Universal Robots URScript: test_regenerated.script

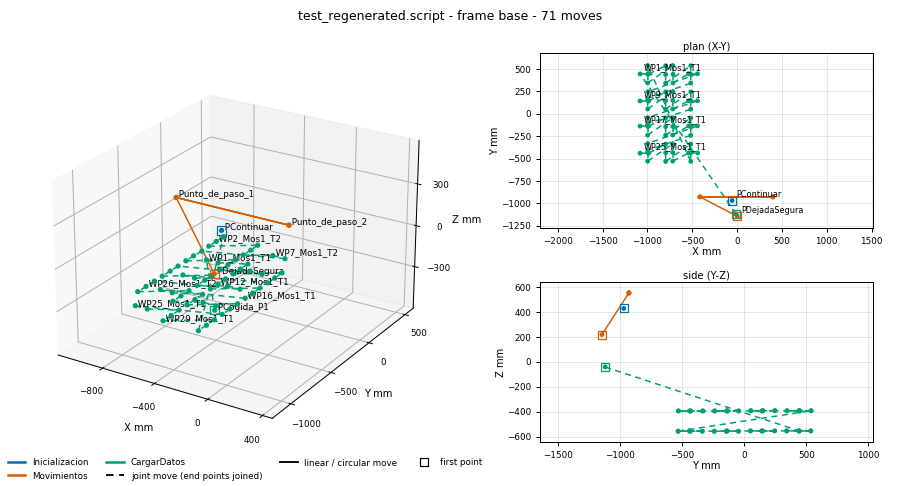
[picture p0: tool path of test_regenerated.script in frame base, 71 of 89 moves have a stored position in this frame; points joined in program order, loops and branches not executed]
def P002_008_L16_REC_AMB_MF():
  set_safety_mode_transition_hardness(1)
  set_tool_communication(False, 115200, 0, 1, 1.5, 3.5)
  set_tool_output_mode(0)
  set_tool_digital_output_mode(0, 1)
  set_tool_digital_output_mode(1, 1)
  set_tool_voltage(24)
  set_tcp(p[0.0,-0.14,0.054,0.0,0.0,0.0])
  set_payload(0.84)
  set_standard_analog_input_domain(0, 1)
  set_standard_analog_input_domain(1, 1)
  set_tool_analog_input_domain(0, 1)
  set_tool_analog_input_domain(1, 1)
  set_analog_outputdomain(0, 0)
  set_analog_outputdomain(1, 0)
  set_input_actions_to_default()
  set_runstate_gp_boolean_output_to_value(15, 3)
  set_gravity([0.0, 0.0, 9.82])
  step_count_91e529f0_9954_4772_b49d_1590ab779229 = 0
  thread Step_Counter_Thread_984ad8c2_81a8_4544_ae12_e3986bad7eaf():
    while (True):
      step_count_91e529f0_9954_4772_b49d_1590ab779229 = step_count_91e529f0_9954_4772_b49d_1590ab779229 + 1
      sync()
    end
  end
  run Step_Counter_Thread_984ad8c2_81a8_4544_ae12_e3986bad7eaf()
  global AlarmaVF2=False
  global ordenM9_T1=[1, 2, 3, 4, 5, 6, 7, 8, 1, 1, 1, 1, 1, 1, 1, 1, 1, 1, 1, 1, 1, 1, 1, 1, 1]
  global AlarmaVF1=False
  global linea=1
  global AlarmaQM2=False
  global LineaHabilitada=[True, True]
  global AlarmaQM1=False
  global ContPrd=0
  global P_Tipo1_Mos9=[p[100, 100, 100, 0, 0, 0], p[100, 100, 100, 0, 0, 0], p[100, 100, 100, 0, 0, 0], p[100, 100, 100, 0, 0, 0], p[100, 100, 100, 0, 0, 0], p[100, 100, 100, 0, 0, 0], p[100, 100, 100, 0, 0, 0], p[100, 100, 100, 0, 0, 0], p[100, 100, 100, 0, 0, 0], p[100, 100, 100, 0, 0, 0], p[100, 100, 100, 0, 0, 0], p[100, 100, 100, 0, 0, 0], p[100, 100, 100, 0, 0, 0], p[100, 100, 100, 0, 0, 0], p[100, 100, 100, 0, 0, 0], p[100, 100, 100, 0, 0, 0], p[100, 100, 100, 0, 0, 0], p[100, 100, 100, 0, 0, 0], p[100, 100, 100, 0, 0, 0], p[100, 100, 100, 0, 0, 0], p[100, 100, 100, 0, 0, 0], p[100, 100, 100, 0, 0, 0], p[100, 100, 100, 0, 0, 0], p[100, 100, 100, 0, 0, 0], p[100, 100, 100, 0, 0, 0]]
  global P_Tipo1_Mos8=[p[100, 100, 100, 0, 0, 0], p[100, 100, 100, 0, 0, 0], p[100, 100, 100, 0, 0, 0], p[100, 100, 100, 0, 0, 0], p[100, 100, 100, 0, 0, 0], p[100, 100, 100, 0, 0, 0], p[100, 100, 100, 0, 0, 0], p[100, 100, 100, 0, 0, 0], p[100, 100, 100, 0, 0, 0], p[100, 100, 100, 0, 0, 0], p[100, 100, 100, 0, 0, 0], p[100, 100, 100, 0, 0, 0], p[100, 100, 100, 0, 0, 0], p[100, 100, 100, 0, 0, 0], p[100, 100, 100, 0, 0, 0], p[100, 100, 100, 0, 0, 0], p[100, 100, 100, 0, 0, 0], p[100, 100, 100, 0, 0, 0], p[100, 100, 100, 0, 0, 0], p[100, 100, 100, 0, 0, 0], p[100, 100, 100, 0, 0, 0], p[100, 100, 100, 0, 0, 0], p[100, 100, 100, 0, 0, 0], p[100, 100, 100, 0, 0, 0], p[100, 100, 100, 0, 0, 0]]
  global P_Tipo1_Mos7=[p[100, 100, 100, 0, 0, 0], p[100, 100, 100, 0, 0, 0], p[100, 100, 100, 0, 0, 0], p[100, 100, 100, 0, 0, 0], p[100, 100, 100, 0, 0, 0], p[100, 100, 100, 0, 0, 0], p[100, 100, 100, 0, 0, 0], p[100, 100, 100, 0, 0, 0], p[100, 100, 100, 0, 0, 0], p[100, 100, 100, 0, 0, 0], p[100, 100, 100, 0, 0, 0], p[100, 100, 100, 0, 0, 0], p[100, 100, 100, 0, 0, 0], p[100, 100, 100, 0, 0, 0], p[100, 100, 100, 0, 0, 0], p[100, 100, 100, 0, 0, 0], p[100, 100, 100, 0, 0, 0], p[100, 100, 100, 0, 0, 0], p[100, 100, 100, 0, 0, 0], p[100, 100, 100, 0, 0, 0], p[100, 100, 100, 0, 0, 0], p[100, 100, 100, 0, 0, 0], p[100, 100, 100, 0, 0, 0], p[100, 100, 100, 0, 0, 0], p[100, 100, 100, 0, 0, 0]]
  global P_Tipo1_Mos6=[p[100, 100, 100, 0, 0, 0], p[100, 100, 100, 0, 0, 0], p[100, 100, 100, 0, 0, 0], p[100, 100, 100, 0, 0, 0], p[100, 100, 100, 0, 0, 0], p[100, 100, 100, 0, 0, 0], p[100, 100, 100, 0, 0, 0], p[100, 100, 100, 0, 0, 0], p[100, 100, 100, 0, 0, 0], p[100, 100, 100, 0, 0, 0], p[100, 100, 100, 0, 0, 0], p[100, 100, 100, 0, 0, 0], p[100, 100, 100, 0, 0, 0], p[100, 100, 100, 0, 0, 0], p[100, 100, 100, 0, 0, 0], p[100, 100, 100, 0, 0, 0], p[100, 100, 100, 0, 0, 0], p[100, 100, 100, 0, 0, 0], p[100, 100, 100, 0, 0, 0], p[100, 100, 100, 0, 0, 0], p[100, 100, 100, 0, 0, 0], p[100, 100, 100, 0, 0, 0], p[100, 100, 100, 0, 0, 0], p[100, 100, 100, 0, 0, 0], p[100, 100, 100, 0, 0, 0]]
  global P_Tipo1_Mos5=[p[100, 100, 100, 0, 0, 0], p[100, 100, 100, 0, 0, 0], p[100, 100, 100, 0, 0, 0], p[100, 100, 100, 0, 0, 0], p[100, 100, 100, 0, 0, 0], p[100, 100, 100, 0, 0, 0], p[100, 100, 100, 0, 0, 0], p[100, 100, 100, 0, 0, 0], p[100, 100, 100, 0, 0, 0], p[100, 100, 100, 0, 0, 0], p[100, 100, 100, 0, 0, 0], p[100, 100, 100, 0, 0, 0], p[100, 100, 100, 0, 0, 0], p[100, 100, 100, 0, 0, 0], p[100, 100, 100, 0, 0, 0], p[100, 100, 100, 0, 0, 0], p[100, 100, 100, 0, 0, 0], p[100, 100, 100, 0, 0, 0], p[100, 100, 100, 0, 0, 0], p[100, 100, 100, 0, 0, 0], p[100, 100, 100, 0, 0, 0], p[100, 100, 100, 0, 0, 0], p[100, 100, 100, 0, 0, 0], p[100, 100, 100, 0, 0, 0], p[100, 100, 100, 0, 0, 0]]
  global P_Tipo1_Mos4=[p[100, 100, 100, 0, 0, 0], p[100, 100, 100, 0, 0, 0], p[100, 100, 100, 0, 0, 0], p[100, 100, 100, 0, 0, 0], p[100, 100, 100, 0, 0, 0], p[100, 100, 100, 0, 0, 0], p[100, 100, 100, 0, 0, 0], p[100, 100, 100, 0, 0, 0], p[100, 100, 100, 0, 0, 0], p[100, 100, 100, 0, 0, 0], p[100, 100, 100, 0, 0, 0], p[100, 100, 100, 0, 0, 0], p[100, 100, 100, 0, 0, 0], p[100, 100, 100, 0, 0, 0], p[100, 100, 100, 0, 0, 0], p[100, 100, 100, 0, 0, 0], p[100, 100, 100, 0, 0, 0], p[100, 100, 100, 0, 0, 0], p[100, 100, 100, 0, 0, 0], p[100, 100, 100, 0, 0, 0], p[100, 100, 100, 0, 0, 0], p[100, 100, 100, 0, 0, 0], p[100, 100, 100, 0, 0, 0], p[100, 100, 100, 0, 0, 0], p[100, 100, 100, 0, 0, 0]]
  global PrdsReq=1
  global P_Tipo1_Mos3=[p[1.16604, 0.55562, 0.63575, 3.14108, -0.00276, -8.40000000000000035E-04], p[0.94603, 0.55481, 0.62022, 3.14109, -0.00285, -8.89999999999999949E-04], p[0.72803, 0.55407, 0.62302, 3.1411, -0.01338, -8.19999999999999982E-04], p[0.511, 0.5552, 0.61604, 3.14122, -0.01324, -8.49999999999999953E-04], p[0.29303, 0.5544, 0.62251, 3.14118, -0.01329, -8.99999999999999975E-04], p[1.00128, 0.17498, 0.62283, 2.22765, -2.21424, -2.30000000000000007E-04], p[0.4544, 0.17301, 0.61254, 2.22767, -2.21422, -2.99999999999999974E-04], p[100, 100, 100, 0, 0, 0], p[100, 100, 100, 0, 0, 0], p[100, 100, 100, 0, 0, 0], p[100, 100, 100, 0, 0, 0], p[100, 100, 100, 0, 0, 0], p[100, 100, 100, 0, 0, 0], p[100, 100, 100, 0, 0, 0], p[100, 100, 100, 0, 0, 0], p[100, 100, 100, 0, 0, 0], p[100, 100, 100, 0, 0, 0], p[100, 100, 100, 0, 0, 0], p[100, 100, 100, 0, 0, 0], p[100, 100, 100, 0, 0, 0], p[100, 100, 100, 0, 0, 0], p[100, 100, 100, 0, 0, 0], p[100, 100, 100, 0, 0, 0], p[100, 100, 100, 0, 0, 0], p[100, 100, 100, 0, 0, 0]]
  global P_Tipo1_Mos2=[p[0.99704, 0.69994, 0.4025, 2.20418, 2.23837, -0.00134], p[0.99871, 0.49941, 0.39482, 2.21365, 2.229, -0.00133], p[0.70631, 0.6015, 0.38963, 0.00568, -3.14107, 0.00118], p[0.50788, 0.60078, 0.39072, 0.00568, -3.14107, 0.00118], p[0.30863, 0.60101, 0.39721, 0.00568, -3.14107, 0.00118], p[0.10677, 0.60171, 0.39277, 0.00568, -3.14107, 0.00118], p[1.0952, 0.20925, 0.39062, 3.14092, 0.00568, -7.10000000000000019E-04], p[0.89523, 0.21023, 0.40246, 3.14092, 0.00568, -7.10000000000000019E-04], p[0.6952, 0.21273, 0.39826, 3.14092, 0.00568, -7.10000000000000019E-04], p[0.49709, 0.21201, 0.39756, 3.14092, 0.00568, -7.10000000000000019E-04], p[0.20516, 0.31346, 0.39069, 2.22486, -2.21683, 2.99999999999999974E-04], p[0.20589, 0.11488, 0.39661, 2.22486, -2.21683, 2.99999999999999974E-04], p[100, 100, 100, 0, 0, 0], p[100, 100, 100, 0, 0, 0], p[100, 100, 100, 0, 0, 0], p[100, 100, 100, 0, 0, 0], p[100, 100, 100, 0, 0, 0], p[100, 100, 100, 0, 0, 0], p[100, 100, 100, 0, 0, 0], p[100, 100, 100, 0, 0, 0], p[100, 100, 100, 0, 0, 0], p[100, 100, 100, 0, 0, 0], p[100, 100, 100, 0, 0, 0], p[100, 100, 100, 0, 0, 0], p[100, 100, 100, 0, 0, 0]]
  global PalletOk=[True, False]
  global P_Tipo1_Mos1=[p[1.04122, 0.73691, 0.32186, -3.1356, -0.00672, -0.01102], p[1.04157, 0.63991, 0.32193, -3.1356, -0.00674, -0.01104], p[1.13376, 0.45174, 0.32215, -2.21965, 2.21023, -0.00123], p[1.03676, 0.45138, 0.32217, -2.21965, 2.21026, -0.00124], p[0.93976, 0.451, 0.3222, -2.21964, 2.21028, -0.00128], p[1.13477, 0.17175, 0.32228, -2.21961, 2.21034, -0.00133], p[1.03777, 0.1714, 0.32233, -2.21962, 2.21032, -0.00135], p[0.94077, 0.17108, 0.32239, -2.21962, 2.21028, -0.00136], p[0.73923, 0.73581, 0.32199, -3.13562, -0.00685, -0.01105], p[0.73959, 0.63882, 0.32205, -3.13564, -0.00684, -0.01107], p[0.84276, 0.45068, 0.32225, -2.21963, 2.21023, -0.00125], p[0.74576, 0.45033, 0.32229, -2.21964, 2.21024, -0.00125], p[0.64876, 0.44998, 0.32233, -2.21967, 2.21024, -0.00121], p[0.84377, 0.17069, 0.32246, -2.2197, 2.21021, -0.00117], p[0.74677, 0.17036, 0.32253, -2.21965, 2.2102, -0.00112], p[0.64977, 0.17002, 0.32257, -2.21967, 2.21018, -0.00108], p[0.45923, 0.73477, 0.32211, -3.13566, -0.00681, -0.01102], p[0.45959, 0.63781, 0.32216, -3.13571, -0.00678, -0.01101], p[0.55176, 0.44964, 0.32025, 2.216, 2.22572, 0.01433], p[0.45476, 0.4493, 0.3203, 2.21603, 2.22569, 0.01434], p[0.35776, 0.44894, 0.32035, 2.21598, 2.22574, 0.01432], p[0.55277, 0.16964, 0.32047, 2.21602, 2.22572, 0.0143], p[0.45577, 0.16927, 0.3205, 2.21599, 2.22573, 0.0143], p[0.35877, 0.16893, 0.32054, 2.21602, 2.2257, 0.0143], p[0.15723, 0.73362, 0.3222, -3.13576, -0.00684, -0.01106]]
  global NPaletTot=5422
  global PalletReady=[True, True]
  global Rec_AltoPrd=[160, 160, 0, 0, 0, 0, 0, 0, 0, 0]
  global P_Tipo2_Mos9=[p[100, 100, 100, 0, 0, 0], p[100, 100, 100, 0, 0, 0], p[100, 100, 100, 0, 0, 0], p[100, 100, 100, 0, 0, 0], p[100, 100, 100, 0, 0, 0], p[100, 100, 100, 0, 0, 0], p[100, 100, 100, 0, 0, 0], p[100, 100, 100, 0, 0, 0], p[100, 100, 100, 0, 0, 0], p[100, 100, 100, 0, 0, 0], p[100, 100, 100, 0, 0, 0], p[100, 100, 100, 0, 0, 0], p[100, 100, 100, 0, 0, 0], p[100, 100, 100, 0, 0, 0], p[100, 100, 100, 0, 0, 0], p[100, 100, 100, 0, 0, 0], p[100, 100, 100, 0, 0, 0], p[100, 100, 100, 0, 0, 0], p[100, 100, 100, 0, 0, 0], p[100, 100, 100, 0, 0, 0], p[100, 100, 100, 0, 0, 0], p[100, 100, 100, 0, 0, 0], p[100, 100, 100, 0, 0, 0], p[100, 100, 100, 0, 0, 0], p[100, 100, 100, 0, 0, 0]]
  global P_Tipo2_Mos8=[p[100, 100, 100, 0, 0, 0], p[100, 100, 100, 0, 0, 0], p[100, 100, 100, 0, 0, 0], p[100, 100, 100, 0, 0, 0], p[100, 100, 100, 0, 0, 0], p[100, 100, 100, 0, 0, 0], p[100, 100, 100, 0, 0, 0], p[100, 100, 100, 0, 0, 0], p[100, 100, 100, 0, 0, 0], p[100, 100, 100, 0, 0, 0], p[100, 100, 100, 0, 0, 0], p[100, 100, 100, 0, 0, 0], p[100, 100, 100, 0, 0, 0], p[100, 100, 100, 0, 0, 0], p[100, 100, 100, 0, 0, 0], p[100, 100, 100, 0, 0, 0], p[100, 100, 100, 0, 0, 0], p[100, 100, 100, 0, 0, 0], p[100, 100, 100, 0, 0, 0], p[100, 100, 100, 0, 0, 0], p[100, 100, 100, 0, 0, 0], p[100, 100, 100, 0, 0, 0], p[100, 100, 100, 0, 0, 0], p[100, 100, 100, 0, 0, 0], p[100, 100, 100, 0, 0, 0]]
  global P_Tipo2_Mos7=[p[100, 100, 100, 0, 0, 0], p[100, 100, 100, 0, 0, 0], p[100, 100, 100, 0, 0, 0], p[100, 100, 100, 0, 0, 0], p[100, 100, 100, 0, 0, 0], p[100, 100, 100, 0, 0, 0], p[100, 100, 100, 0, 0, 0], p[100, 100, 100, 0, 0, 0], p[100, 100, 100, 0, 0, 0], p[100, 100, 100, 0, 0, 0], p[100, 100, 100, 0, 0, 0], p[100, 100, 100, 0, 0, 0], p[100, 100, 100, 0, 0, 0], p[100, 100, 100, 0, 0, 0], p[100, 100, 100, 0, 0, 0], p[100, 100, 100, 0, 0, 0], p[100, 100, 100, 0, 0, 0], p[100, 100, 100, 0, 0, 0], p[100, 100, 100, 0, 0, 0], p[100, 100, 100, 0, 0, 0], p[100, 100, 100, 0, 0, 0], p[100, 100, 100, 0, 0, 0], p[100, 100, 100, 0, 0, 0], p[100, 100, 100, 0, 0, 0], p[100, 100, 100, 0, 0, 0]]
  global P_Tipo2_Mos6=[p[100, 100, 100, 0, 0, 0], p[100, 100, 100, 0, 0, 0], p[100, 100, 100, 0, 0, 0], p[100, 100, 100, 0, 0, 0], p[100, 100, 100, 0, 0, 0], p[100, 100, 100, 0, 0, 0], p[100, 100, 100, 0, 0, 0], p[100, 100, 100, 0, 0, 0], p[100, 100, 100, 0, 0, 0], p[100, 100, 100, 0, 0, 0], p[100, 100, 100, 0, 0, 0], p[100, 100, 100, 0, 0, 0], p[100, 100, 100, 0, 0, 0], p[100, 100, 100, 0, 0, 0], p[100, 100, 100, 0, 0, 0], p[100, 100, 100, 0, 0, 0], p[100, 100, 100, 0, 0, 0], p[100, 100, 100, 0, 0, 0], p[100, 100, 100, 0, 0, 0], p[100, 100, 100, 0, 0, 0], p[100, 100, 100, 0, 0, 0], p[100, 100, 100, 0, 0, 0], p[100, 100, 100, 0, 0, 0], p[100, 100, 100, 0, 0, 0], p[100, 100, 100, 0, 0, 0]]
  global P_Tipo2_Mos5=[p[100, 100, 100, 0, 0, 0], p[100, 100, 100, 0, 0, 0], p[100, 100, 100, 0, 0, 0], p[100, 100, 100, 0, 0, 0], p[100, 100, 100, 0, 0, 0], p[100, 100, 100, 0, 0, 0], p[100, 100, 100, 0, 0, 0], p[100, 100, 100, 0, 0, 0], p[100, 100, 100, 0, 0, 0], p[100, 100, 100, 0, 0, 0], p[100, 100, 100, 0, 0, 0], p[100, 100, 100, 0, 0, 0], p[100, 100, 100, 0, 0, 0], p[100, 100, 100, 0, 0, 0], p[100, 100, 100, 0, 0, 0], p[100, 100, 100, 0, 0, 0], p[100, 100, 100, 0, 0, 0], p[100, 100, 100, 0, 0, 0], p[100, 100, 100, 0, 0, 0], p[100, 100, 100, 0, 0, 0], p[100, 100, 100, 0, 0, 0], p[100, 100, 100, 0, 0, 0], p[100, 100, 100, 0, 0, 0], p[100, 100, 100, 0, 0, 0], p[100, 100, 100, 0, 0, 0]]
  global NCapaAct=[1, 1]
  global P_Tipo2_Mos4=[p[100, 100, 100, 0, 0, 0], p[100, 100, 100, 0, 0, 0], p[100, 100, 100, 0, 0, 0], p[100, 100, 100, 0, 0, 0], p[100, 100, 100, 0, 0, 0], p[100, 100, 100, 0, 0, 0], p[100, 100, 100, 0, 0, 0], p[100, 100, 100, 0, 0, 0], p[100, 100, 100, 0, 0, 0], p[100, 100, 100, 0, 0, 0], p[100, 100, 100, 0, 0, 0], p[100, 100, 100, 0, 0, 0], p[100, 100, 100, 0, 0, 0], p[100, 100, 100, 0, 0, 0], p[100, 100, 100, 0, 0, 0], p[100, 100, 100, 0, 0, 0], p[100, 100, 100, 0, 0, 0], p[100, 100, 100, 0, 0, 0], p[100, 100, 100, 0, 0, 0], p[100, 100, 100, 0, 0, 0], p[100, 100, 100, 0, 0, 0], p[100, 100, 100, 0, 0, 0], p[100, 100, 100, 0, 0, 0], p[100, 100, 100, 0, 0, 0], p[100, 100, 100, 0, 0, 0]]
  global P_Tipo2_Mos3=[p[1.00663, 0.71329, 0.77118, 2.22767, -2.21422, -2.99999999999999974E-04], p[0.45784, 0.71261, 0.76931, 2.22767, -2.21422, -2.99999999999999974E-04], p[1.16656, 0.33923, 0.80534, 3.1413, -0.00972, -9.60000000000000024E-04], p[0.9489, 0.33841, 0.79064, 3.14125, -0.01511, -0.00113], p[0.73088, 0.33763, 0.77696, 3.14125, -0.01511, -0.00115], p[0.5119, 0.33683, 0.78134, 3.14126, -0.01514, -0.00122], p[0.29291, 0.33753, 0.79002, 3.14126, -0.0151, -0.00118], p[100, 100, 100, 0, 0, 0], p[100, 100, 100, 0, 0, 0], p[100, 100, 100, 0, 0, 0], p[100, 100, 100, 0, 0, 0], p[100, 100, 100, 0, 0, 0], p[100, 100, 100, 0, 0, 0], p[100, 100, 100, 0, 0, 0], p[100, 100, 100, 0, 0, 0], p[100, 100, 100, 0, 0, 0], p[100, 100, 100, 0, 0, 0], p[100, 100, 100, 0, 0, 0], p[100, 100, 100, 0, 0, 0], p[100, 100, 100, 0, 0, 0], p[100, 100, 100, 0, 0, 0], p[100, 100, 100, 0, 0, 0], p[100, 100, 100, 0, 0, 0], p[100, 100, 100, 0, 0, 0], p[100, 100, 100, 0, 0, 0]]
  global P_Tipo2_Mos2=[p[1.09673, 0.60531, 0.52579, 0.00568, -3.14105, 0.00108], p[0.89826, 0.60459, 0.53036, 0.00568, -3.14105, 0.00108], p[0.69753, 0.60155, 0.53003, 0.00568, -3.14105, 0.00108], p[0.49739, 0.60082, 0.52062, 0.00568, -3.14105, 0.00108], p[0.20624, 0.7039, 0.53456, 2.22483, -2.21679, 2.70000000000000003E-04], p[0.2033, 0.50369, 0.53493, 2.22483, -2.21679, 2.70000000000000003E-04], p[1.00083, 0.30839, 0.52599, 2.21734, 2.22537, -0.00119], p[1.00155, 0.11082, 0.53432, 2.21734, 2.22537, -0.00119], p[0.70593, 0.21094, 0.5328, 3.14079, 0.00568, -6.59999999999999996E-04], p[0.50462, 0.2113, 0.536, 3.14079, 0.00568, -6.59999999999999996E-04], p[0.30453, 0.20978, 0.53196, 3.14079, 0.00568, -6.59999999999999996E-04], p[0.10494, 0.20881, 0.53476, 3.14079, 0.00568, -6.59999999999999996E-04], p[100, 100, 100, 0, 0, 0], p[100, 100, 100, 0, 0, 0], p[100, 100, 100, 0, 0, 0], p[100, 100, 100, 0, 0, 0], p[100, 100, 100, 0, 0, 0], p[100, 100, 100, 0, 0, 0], p[100, 100, 100, 0, 0, 0], p[100, 100, 100, 0, 0, 0], p[100, 100, 100, 0, 0, 0], p[100, 100, 100, 0, 0, 0], p[100, 100, 100, 0, 0, 0], p[100, 100, 100, 0, 0, 0], p[100, 100, 100, 0, 0, 0]]
  global Rec_LargoPrd=[280, 280, 0, 0, 0, 0, 0, 0, 0, 0]
  global P_Tipo2_Mos1=[p[1.13563, 0.65237, 0.48446, -2.21948, 2.21033, -0.00109], p[1.03864, 0.65202, 0.48456, -2.21938, 2.21038, -0.00105], p[0.94165, 0.65167, 0.48455, -2.21934, 2.21059, -0.00125], p[1.13664, 0.37237, 0.48466, -2.21936, 2.21046, -0.00115], p[1.03965, 0.36896, 0.4847, -2.21936, 2.2105, -0.00107], p[0.94264, 0.3697, 0.48478, -2.21931, 2.21043, -0.00116], p[1.0458, 0.19393, 0.48294, -0.0066, 3.13445, 0.00964], p[1.04614, 0.09604, 0.48297, -0.00652, 3.13457, 0.00962], p[0.84463, 0.64649, 0.48465, -2.21937, 2.21047, -0.00112], p[0.74763, 0.65096, 0.48472, -2.21939, 2.21045, -0.00115], p[0.65062, 0.65008, 0.48479, -2.21938, 2.21038, -0.00104], p[0.84564, 0.37132, 0.48489, -2.21934, 2.21043, -0.00103], p[0.74863, 0.3709, 0.48492, -2.21942, 2.21043, -0.00105], p[0.65165, 0.37061, 0.48497, -2.21941, 2.2104, -0.001], p[0.74377, 0.19295, 0.48309, -0.00655, 3.13449, 0.00967], p[0.74414, 0.09495, 0.48316, -0.00643, 3.13452, 0.00969], p[0.55354, 0.65026, 0.48282, 2.21558, 2.22646, 0.01462], p[0.45664, 0.64991, 0.4828, 2.21568, 2.22629, 0.01454], p[0.35961, 0.64956, 0.48289, 2.21567, 2.22635, 0.01466], p[0.55461, 0.36988, 0.48306, 2.21569, 2.22642, 0.01467], p[0.45764, 0.36991, 0.48313, 2.21578, 2.22639, 0.0147], p[0.36063, 0.36956, 0.48318, 2.2158, 2.22641, 0.01483], p[0.46379, 0.19193, 0.4832, -0.00647, 3.13448, 0.00958], p[0.4641, 0.09393, 0.4833, -0.00651, 3.13456, 0.00968], p[0.2656, 0.64922, 0.48297, 2.21575, 2.22631, 0.01469]]
  global Movs2en2_M10_T2=[False, False, False, False, False, False, False, False, False, False, False, False, False, False, False, False, False, False, False, False, False, False, False, False, False]
  global P_Tipo2_Mos10=[p[100, 100, 100, 0, 0, 0], p[100, 100, 100, 0, 0, 0], p[100, 100, 100, 0, 0, 0], p[100, 100, 100, 0, 0, 0], p[100, 100, 100, 0, 0, 0], p[100, 100, 100, 0, 0, 0], p[100, 100, 100, 0, 0, 0], p[100, 100, 100, 0, 0, 0], p[100, 100, 100, 0, 0, 0], p[100, 100, 100, 0, 0, 0], p[100, 100, 100, 0, 0, 0], p[100, 100, 100, 0, 0, 0], p[100, 100, 100, 0, 0, 0], p[100, 100, 100, 0, 0, 0], p[100, 100, 100, 0, 0, 0], p[100, 100, 100, 0, 0, 0], p[100, 100, 100, 0, 0, 0], p[100, 100, 100, 0, 0, 0], p[100, 100, 100, 0, 0, 0], p[100, 100, 100, 0, 0, 0], p[100, 100, 100, 0, 0, 0], p[100, 100, 100, 0, 0, 0], p[100, 100, 100, 0, 0, 0], p[100, 100, 100, 0, 0, 0], p[100, 100, 100, 0, 0, 0]]
  global Movs2en2_M10_T1=[False, False, False, False, False, False, False, False, False, False, False, False, False, False, False, False, False, False, False, False, False, False, False, False, False]
  global Rec_AnchoPrd=[97, 97, 0, 0, 0, 0, 0, 0, 0, 0]
  global umbral_bajada=515
  global pos_subida=[0, 0]
  global PuntosCogida=[p[-0.01294, -1.11748, -0.04056, -2.21361, -2.21498, -9.60000000000000024E-04], p[-0.01294, -1.11748, -0.04056, -2.21361, -2.21498, -9.60000000000000024E-04], p[-0.01294, -1.11748, -0.04056, -2.21361, -2.21498, -9.60000000000000024E-04], p[100, 100, 100, 0, 0, 0], p[100, 100, 100, 0, 0, 0], p[100, 100, 100, 0, 0, 0], p[100, 100, 100, 0, 0, 0], p[100, 100, 100, 0, 0, 0], p[100, 100, 100, 0, 0, 0], p[100, 100, 100, 0, 0, 0], p[100, 100, 100, 0, 0, 0], p[100, 100, 100, 0, 0, 0], p[100, 100, 100, 0, 0, 0], p[100, 100, 100, 0, 0, 0], p[100, 100, 100, 0, 0, 0]]
  global AltoBaseRobot=885
  global Rec_TipoCapa=[1, 2, 1, 2, 1, 2, 1, 2, 1, 2, 1, 2, 1, 2, 1, 2, 1, 2, 1, 2, 1, 2, 1, 2, 1, 2, 1, 2, 1, 2]
  global payload=1.1
  global P_Tipo1_Mos10=[p[100, 100, 100, 0, 0, 0], p[100, 100, 100, 0, 0, 0], p[100, 100, 100, 0, 0, 0], p[100, 100, 100, 0, 0, 0], p[100, 100, 100, 0, 0, 0], p[100, 100, 100, 0, 0, 0], p[100, 100, 100, 0, 0, 0], p[100, 100, 100, 0, 0, 0], p[100, 100, 100, 0, 0, 0], p[100, 100, 100, 0, 0, 0], p[100, 100, 100, 0, 0, 0], p[100, 100, 100, 0, 0, 0], p[100, 100, 100, 0, 0, 0], p[100, 100, 100, 0, 0, 0], p[100, 100, 100, 0, 0, 0], p[100, 100, 100, 0, 0, 0], p[100, 100, 100, 0, 0, 0], p[100, 100, 100, 0, 0, 0], p[100, 100, 100, 0, 0, 0], p[100, 100, 100, 0, 0, 0], p[100, 100, 100, 0, 0, 0], p[100, 100, 100, 0, 0, 0], p[100, 100, 100, 0, 0, 0], p[100, 100, 100, 0, 0, 0], p[100, 100, 100, 0, 0, 0]]
  global CartonBase=[False, False]
  global Aprox=[0, 0, 0, 0, 0, 0, 0, 0, 0, 0, 0, 0, 0, 0, 0, 0]
  global Rec_2Vacios=[False, False, False, False, False, False, False, False, False, False]
  global oEV4=False
  global LineaPreparada=[False, False]
  global oEV2=False
  global oEV1=False
  global NMovAct=[18, 1]
  global Rec_Cogida2en2=[False, False, False, False, False, False, False, False, False, False]
  global AltoPalet=155
  global reset_puntos=False
  global PonerCarton=[False, False]
  global Alarma=False
  global Programa=1
  global M_PL=False
  global ManoConProd=False
  global ManoConCarton=False
  global Rec_PesoPrd=[1.23, 1.23, 0.0, 0.0, 0.0, 0.0, 0.0, 0.0, 0.0, 0.0]
  global ordenM10_T2=[1, 2, 3, 4, 5, 6, 7, 8, 1, 1, 1, 1, 1, 1, 1, 1, 1, 1, 1, 1, 1, 1, 1, 1, 1]
  global ordenM10_T1=[1, 2, 3, 4, 5, 6, 7, 8, 1, 1, 1, 1, 1, 1, 1, 1, 1, 1, 1, 1, 1, 1, 1, 1, 1]
  global NPaletAct=3962
  global pos_objetivo=p[0.26485, -1.11984, -0.10292, -2.09801, 2.08938, -0.25492]
  global AlarmaVacio=False
  global Movs2en2_M1_T2=[False, False, False, False, False, False, False, False, False, False, False, False, False, False, False, False, False, False, False, False, False, False, False, False, False]
  global Movs2en2_M1_T1=[False, False, False, False, False, False, False, False, False, False, False, False, False, False, False, False, False, False, False, False, False, False, False, False, False]
  global PalletEnd=[False, True]
  global ordenM1_T2=[8, 7, 4, 5, 6, 1, 2, 3, 16, 15, 12, 13, 14, 9, 10, 11, 24, 23, 20, 21, 22, 17, 18, 19, 32]
  global ordenM1_T1=[6, 7, 8, 3, 4, 5, 2, 1, 14, 15, 16, 11, 12, 13, 10, 9, 22, 23, 24, 19, 20, 21, 18, 17, 30]
  global Movs2en2_M2_T2=[False, False, False, False, False, False, False, False, False, False, False, False, False, False, False, False, False, False, False, False, False, False, False, False, False]
  global Movs2en2_M2_T1=[False, False, False, False, False, False, False, False, False, False, False, False, False, False, False, False, False, False, False, False, False, False, False, False, False]
  global ordenM2_T2=[8, 7, 9, 10, 11, 12, 1, 2, 3, 4, 6, 5, 1, 1, 1, 1, 1, 1, 1, 1, 1, 1, 1, 1, 1]
  global Rec_Carton=[False, False, False, False, False, False, False, False, False, False]
  global ordenM2_T1=[7, 8, 9, 10, 12, 11, 2, 1, 3, 4, 5, 6, 1, 1, 1, 1, 1, 1, 1, 1, 1, 1, 1, 1, 1]
  global Movs2en2_M3_T2=[False, False, False, False, False, False, False, False, False, False, False, False, False, False, False, False, False, False, False, False, False, False, False, False, False]
  global Programa_1=2
  global Movs2en2_M3_T1=[False, False, False, False, False, False, False, False, False, False, False, False, False, False, False, False, False, False, False, False, False, False, False, False, False]
  global Rec_NMovsCapa=[32, 32, 0, 0, 0, 0, 0, 0, 0, 0]
  global ordenM3_T2=[3, 4, 5, 6, 7, 1, 2, 1, 1, 1, 1, 1, 1, 1, 1, 1, 1, 1, 1, 1, 1, 1, 1, 1, 1]
  global ordenM3_T1=[6, 7, 1, 2, 3, 4, 5, 1, 1, 1, 1, 1, 1, 1, 1, 1, 1, 1, 1, 1, 1, 1, 1, 1, 1]
  global Movs2en2_M4_T2=[False, False, False, False, False, False, False, False, False, False, False, False, False, False, False, False, False, False, False, False, False, False, False, False, False]
  global Movs2en2_M4_T1=[False, False, False, False, False, False, False, False, False, False, False, False, False, False, False, False, False, False, False, False, False, False, False, False, False]
  global Rec_NCapasTot=[6, 7, 0, 0, 0, 0, 0, 0, 0, 0]
  global ordenM4_T2=[1, 2, 3, 4, 5, 6, 7, 8, 1, 1, 1, 1, 1, 1, 1, 1, 1, 1, 1, 1, 1, 1, 1, 1, 1]
  global Rec_CapasTrab=[True, True, True, False, False, False, False, False, False, False]
  global ProdListo=False
  global ordenM4_T1=[1, 2, 3, 4, 5, 6, 7, 8, 1, 1, 1, 1, 1, 1, 1, 1, 1, 1, 1, 1, 1, 1, 1, 1, 1]
  global Movs2en2_M5_T2=[False, False, False, False, False, False, False, False, False, False, False, False, False, False, False, False, False, False, False, False, False, False, False, False, False]
  global Movs2en2_M5_T1=[False, False, False, False, False, False, False, False, False, False, False, False, False, False, False, False, False, False, False, False, False, False, False, False, False]
  global ordenM5_T2=[1, 2, 3, 4, 5, 6, 7, 8, 1, 1, 1, 1, 1, 1, 1, 1, 1, 1, 1, 1, 1, 1, 1, 1, 1]
  global ordenM5_T1=[1, 2, 3, 4, 5, 6, 7, 8, 1, 1, 1, 1, 1, 1, 1, 1, 1, 1, 1, 1, 1, 1, 1, 1, 1]
  global Movs2en2_M6_T2=[False, False, False, False, False, False, False, False, False, False, False, False, False, False, False, False, False, False, False, False, False, False, False, False, False]
  global Movs2en2_M6_T1=[False, False, False, False, False, False, False, False, False, False, False, False, False, False, False, False, False, False, False, False, False, False, False, False, False]
  global ordenM6_T2=[1, 2, 3, 4, 5, 6, 7, 8, 1, 1, 1, 1, 1, 1, 1, 1, 1, 1, 1, 1, 1, 1, 1, 1, 1]
  global AnchoPalet=800
  global ordenM6_T1=[1, 2, 3, 4, 5, 6, 7, 8, 1, 1, 1, 1, 1, 1, 1, 1, 1, 1, 1, 1, 1, 1, 1, 1, 1]
  global Movs2en2_M7_T2=[False, False, False, False, False, False, False, False, False, False, False, False, False, False, False, False, False, False, False, False, False, False, False, False, False]
  global pos_bajada=[0, 0]
  global Movs2en2_M7_T1=[False, False, False, False, False, False, False, False, False, False, False, False, False, False, False, False, False, False, False, False, False, False, False, False, False]
  global ResetAlarmas=False
  global ordenM7_T2=[1, 2, 3, 4, 5, 6, 7, 8, 1, 1, 1, 1, 1, 1, 1, 1, 1, 1, 1, 1, 1, 1, 1, 1, 1]
  global NPrdAct=[1, 1]
  global Movs2en2_M8_T2=[False, False, False, False, False, False, False, False, False, False, False, False, False, False, False, False, False, False, False, False, False, False, False, False, False]
  global ordenM7_T1=[1, 2, 3, 4, 5, 6, 7, 8, 1, 1, 1, 1, 1, 1, 1, 1, 1, 1, 1, 1, 1, 1, 1, 1, 1]
  global Movs2en2_M8_T1=[False, False, False, False, False, False, False, False, False, False, False, False, False, False, False, False, False, False, False, False, False, False, False, False, False]
  global AltoTransporte=680
  global Rec_Mosaico=[1, 1, 0, 0, 0, 0, 0, 0, 0, 0]
  global ordenM8_T2=[1, 2, 3, 4, 5, 6, 7, 8, 1, 1, 1, 1, 1, 1, 1, 1, 1, 1, 1, 1, 1, 1, 1, 1, 1]
  global ordenM8_T1=[1, 2, 3, 4, 5, 6, 7, 8, 1, 1, 1, 1, 1, 1, 1, 1, 1, 1, 1, 1, 1, 1, 1, 1, 1]
  global Movs2en2_M9_T2=[False, False, False, False, False, False, False, False, False, False, False, False, False, False, False, False, False, False, False, False, False, False, False, False, False]
  global Movs2en2_M9_T1=[False, False, False, False, False, False, False, False, False, False, False, False, False, False, False, False, False, False, False, False, False, False, False, False, False]
  global PSegAtras=p[0.007716780405957183,0.9365680771484418,0.6088949059182273,-1.5709669316014583,1.8546757310268662E-4,1.2933138056551383E-4]
  global PSegDer=p[-1.3409244425804514,0.083036323608216,0.48123901688998855,-1.2719670689283105,-1.163229788032182,1.224260502195706]
  global PSegIzq=p[1.340084782198209,-0.177902950396446,0.33899221418014425,-1.171104712667188,1.2513964548728496,-1.1683450977271492]
  global PSegPickUp=p[-0.04899381203365097,-1.1642098362887696,0.5324100249885306,-0.0554334453004588,-2.23265336008919,2.134801320285594]
  global wObjDejadaRef=p[-0.3500863019098047, -0.5987226873651141, -0.8779278611891395, 9.42972933224836747E-04, 1.63784070804397599E-04, 1.5671793604966087]
  global wobjDejadaRef=p[-0.3500608235485929,-0.598703534451815,-0.8779553249182175,2.683853195153339,-1.6329407514614793,3.4388935169646775E-5]
  # begin: URCap Installation Node
  #   Source: HMI_FranciscoAragon, 4.0.0, Geniotic Solutions SL
  #   Type: HMI
  # end: URCap Installation Node
  global Arranque_from_p=p[-.413745024855, -.280268034161, .401095205191, 2.902434303719, -1.202278191569, .000021368141]
  global Arranque_to_p=p[-.413755691927, -.280260433532, .401096693735, 2.902440840405, -1.202259035281, -.000056728081]
  global PDejadaSegura_p=p[.002715171455, -1.143669533313, .219963206371, -2.213607190275, -2.214979246151, -.000955509289]
  global PDejadaSegura_q=[-1.2953688852883793, -2.4640730802768185, -0.9876246344336348, -1.269355999886388, 1.5621624808640124, 1.8461742949527784]
  global Punto_de_paso_1_p=p[-.415075939126, -.926322746418, .554971813004, -1.273146432212, -2.861989386414, -.006556073600]
  global Punto_de_paso_1_q=[-1.7310930993122886, -1.873788536052527, -1.336793128096824, -1.5077595885815454, 1.5597203717114299, 0.6784194102436473]
  global Punto_de_paso_2_p=p[.399812458066, -.926927515157, .555000000030, 1.201802570685, -2.899078315327, -.014881112522]
  global Punto_de_paso_2_q=[-1.0244784972105911, -1.8614801482241523, -1.3497636848456889, -1.5105610655909203, 1.565811724178163, -0.2380579999078858]
  global Home_p=p[-.055703615062, -.967595028813, .430598506015, .195128277210, -3.124071103987, -.001665921395]
  global Home_q=[-1.446930233632223, -1.817273279229635, -1.6329717636108398, -1.263462857609131, 1.556671142578125, 5.551115123125783E-17]
  global PPerchCogidaCar_p=p[.010116577127, -1.153430844518, .094590411744, -.046099547411, 3.141195381271, -.000298477174]
  global PPerchCogidaCar_q=[-1.4100163618670862, -2.5525084934630335, -1.052506923675537, -1.107565776710846, 1.5683655738830566, 0.13021214306354523]
  global PCogidaCarton_p=p[.264846204336, -1.119836457785, -.102923732977, -2.098006206258, 2.089378388183, -.254921434385]
  global PCogidaCarton_q=[-1.219926659260885, -2.7496749363341273, -1.0751527547836304, -0.8035006088069458, 1.7948288917541504, -1.216395680104391]
  global PDejadaCarton_p=p[-.750395952325, .473204354478, -.777503218896, .020496391888, -3.141493897005, .000057902978]
  global PDejadaCarton_q=[-3.5061636606799524, -3.557664533654684, -0.8158471584320068, -0.339249925022461, 1.5696253776550293, -1.9507959524737757]
  global PIntermedio_p=p[-.004454611980, -1.140193448808, .333338150649, -.046304151311, 3.141167821431, -.000558672612]
  global PIntermedio_q=[-1.4208996931659144, -2.381580492059225, -0.9329356551170349, -1.3978987795165558, 1.568293571472168, 0.11983348429203033]
  global PCogida_P1_p=p[-.012938049433, -1.117475798500, -.040556576898, -2.213607171749, -2.214979239179, -.000955484338]
  global PCogida_P1_q=[-1.3025226126260652, -2.6418259874795638, -1.1471770164608266, -0.9320122391530585, 1.5624976791528353, 1.8380069263771917]
  global WP1_Mos1_T1_p=p[-1.083000000000, .444995617736, -.555031222987, -2.213605874023, -2.215082527224, -.000978759292]
  global WP1_Mos1_T1_q=[-3.414994238416195, -3.2762020582787597, -0.8817537176977259, -0.545512557540123, 1.5618679522456322, -0.27639867593190814]
  global WP2_Mos1_T1_p=p[-.986000000074, .444990562609, -.555031282016, -2.213588110478, -2.215090987381, -.000994015174]
  global WP2_Mos1_T1_q=[-3.443066896336911, -3.200335707781061, -1.1392245980494673, -0.3637585699778292, 1.562699042223965, -0.3043978563837362]
  global WP3_Mos1_T1_p=p[-.797499999948, .536499999948, -.554899597249, -3.134011886263, -.000994831276, .010400379954]
  global WP3_Mos1_T1_q=[-3.406545842022289, -3.1649793447584496, -1.2986759940286152, -0.23987261704319174, 1.562784755792402, 1.3030414708277067]
  global WP4_Mos1_T1_p=p[-.797490936602, .439500000049, -.554926093030, -3.134024962530, -.000972814065, .010360446096]
  global WP4_Mos1_T1_q=[-3.2951543767865425, -3.1509329194263342, -1.3836868677892706, -0.1696041325055413, 1.5621262591810747, 1.4144990554065402]
  global WP5_Mos1_T1_p=p[-.797457474888, .342500000074, -.554947278644, -3.134008876204, -.000953681814, .010331958746]
  global WP5_Mos1_T1_q=[-3.1769796471834715, -3.1434529529812054, -1.4437399023399164, -0.11786127940792479, 1.5614146956250348, 1.5327291700760064]
  global WP6_Mos1_T1_p=p[-.517499999924, .536500000053, -.554962903360, -3.134008794703, -.000887256228, .010266053534]
  global WP6_Mos1_T1_q=[-3.5255687343052045, -3.152668137160764, -1.7441792947373358, 0.19383557141115365, 1.5650973690653858, 1.1844844529224396]
  global WP7_Mos1_T1_p=p[-.517504001451, .439500000074, -.554962933077, -3.133990046014, -.000910870533, .010257170027]
  global WP7_Mos1_T1_q=[-3.3708732832155035, -3.1744454284105794, -1.8230815784612648, 0.2937063230443434, 1.5640146608501548, 1.3392756507817152]
  global WP8_Mos1_T1_p=p[-.517533088052, .342500000074, -.554950285805, -3.133971137405, -.000939119034, .010281014929]
  global WP8_Mos1_T1_q=[-3.1955048488983997, -3.1982663871284567, -1.879667888818024, 0.37297797803095845, 1.5628611989967869, 1.5147202786741782]
  global WP9_Mos1_T1_p=p[-1.082995115837, .142999999899, -.555049486766, -2.213512438716, -2.215173643942, -.001020055055]
  global WP9_Mos1_T1_q=[-3.108487713855308, -3.1986920420288083, -1.1445286743763647, -0.3623024667176704, 1.5601656831388864, 0.03011561399415277]
  global WP10_Mos1_T1_p=p[-.986000000075, .143014489008, -.555063709467, -2.213518649655, -2.215173226723, -.001050683610]
  global WP10_Mos1_T1_q=[-3.104690056910966, -3.1526565771230266, -1.3703002518058094, -0.18261486847237407, 1.560726707112723, 0.03403476645041017]
  global WP11_Mos1_T1_p=p[-.797492743129, .245500000074, -.554938223332, -3.133993482738, -.000981673048, .010396790007]
  global WP11_Mos1_T1_q=[-3.054698186454996, -3.1399670593546847, -1.480065745492647, -0.08592498698683215, 1.5607160051001865, 1.655023044652268]
  global WP12_Mos1_T1_p=p[-.797491829227, .148500000074, -.554947151197, -3.134007035872, -.000986782198, .010380382055]
  global WP12_Mos1_T1_q=[-2.9317491532147715, -3.138805831779737, -1.493391152914974, -0.07480877736613945, 1.5600983421960744, 1.7779840566493752]
  global WP13_Mos1_T1_p=p[-.797494243839, .051500000074, -.554955517335, -3.134041519779, -.001003094448, .010385356496]
  global WP13_Mos1_T1_q=[-2.8118093279764937, -3.1393059396936067, -1.4838713423719936, -0.08489912517565656, 1.5595755432836607, 1.8979118288205115]
  global WP14_Mos1_T1_p=p[-.517499999990, .245500000007, -.554932243017, -3.134052867863, -.001045261146, .010412524902]
  global WP14_Mos1_T1_q=[-3.005884253661509, -3.217114603722517, -1.9143364486632244, 0.42510103404604876, 1.5618644278210367, 1.704340593737917]
  global WP15_Mos1_T1_p=p[-.517521017766, .148500000074, -.554912384222, -3.134050907913, -.001019358102, .010487844170]
  global WP15_Mos1_T1_q=[-2.8136778516979484, -3.224730713208515, -1.927147803361751, 0.4438767493599401, 1.5609779447057939, 1.8965946779462701]
  global WP16_Mos1_T1_p=p[-.517528672925, .051500000042, -.554914438302, -3.134062797292, -.001046663677, .010522724593]
  global WP16_Mos1_T1_q=[-2.6327614820179117, -3.218449238746127, -1.9182810151452774, 0.4270216170294319, 1.5603894732193924, 2.077484090881873]
  global WP17_Mos1_T1_p=p[-1.082961866822, -.136999999979, -.555067507355, -2.213575177365, -2.215176616537, -.001038536040]
  global WP17_Mos1_T1_q=[-2.8132576690394613, -3.1978275687863666, -1.146527400057824, -0.3637339080507651, 1.5586776781411618, 0.3253881858363455]
  global WP18_Mos1_T1_p=p[-.986000000062, -.136985288371, -.555087652244, -2.213615671018, -2.215183846961, -.001084878352]
  global WP18_Mos1_T1_q=[-2.776129922085309, -3.1519210777119473, -1.3721213805337262, -0.18443536535564586, 1.5591559131269075, 0.362650497336826]
  global WP19_Mos1_T1_p=p[-.797500000000, -.045500000011, -.557089378695, .001194163262, -3.134979492236, -.011780656361]
  global WP19_Mos1_T1_q=[-3.0407506051743916, -3.1398229420730015, -1.4822846736943642, -0.08400067286175084, 1.5607105933928371, -1.472754823848132]
  global WP20_Mos1_T1_p=p[-.797509234577, -.142499999926, -.557087429393, .001152230494, -3.134974589154, -.011786075227]
  global WP20_Mos1_T1_q=[-2.9179880928177813, -3.1388478395232196, -1.4930209525591893, -0.07527473882170543, 1.560084930232145, -1.3499523789318726]
  global WP21_Mos1_T1_p=p[-.797499123300, -.239499999935, -.557081160798, .001219107401, -3.134985635375, -.011772633060]
  global WP21_Mos1_T1_q=[-2.798633613642949, -3.1395332886650777, -1.4809271413736251, -0.08777016197674925, 1.559553540370999, -1.230644041158535]
  global WP22_Mos1_T1_p=p[-.517499999998, -.045499999998, -.557068708462, .001176816811, -3.134981585240, -.011744862049]
  global WP22_Mos1_T1_q=[-2.9840147592453734, -3.218530222375638, -1.9165924582237412, 0.42853862536203347, 1.5617903035805643, -1.4154610132470928]
  global WP23_Mos1_T1_p=p[-.517485376195, -.142499999926, -.557082745401, .001202726494, -3.134991904859, -.011756353316]
  global WP23_Mos1_T1_q=[-2.7924640981655093, -3.2246700440434783, -1.9269303613909763, 0.4433023338471797, 1.560957675202731, -1.2238999684244014]
  global WP24_Mos1_T1_p=p[-.517488842705, -.239499999926, -.557086444522, .001159303464, -3.134994449771, -.011757487852]
  global WP24_Mos1_T1_q=[-2.6136550319137317, -3.2168642335641784, -1.915598885890863, 0.4224521449347018, 1.5604191950525717, -1.0450773167382001]
  global WP25_Mos1_T1_p=p[-1.082905598438, -.439000000090, -.555136347116, -2.213587104467, -2.215234134382, -.001176142602]
  global WP25_Mos1_T1_q=[-2.537187044583862, -3.2729547766914457, -0.8889045380033389, -0.5489898293785336, 1.5574061210945054, 0.6013774591411077]
  global WP26_Mos1_T1_p=p[-.986000000039, -.439010467011, -.555101090818, -2.213582376621, -2.215255508308, -.001108594343]
  global WP26_Mos1_T1_q=[-2.4787775760283552, -3.1976992119202348, -1.1452224176205483, -0.3684682511940238, 1.5579796540448014, 0.6598607798566604]
  global WP27_Mos1_T1_p=p[-.797479794138, -.336499999926, -.557088459181, .001271270436, -3.135008829694, -.011740450862]
  global WP27_Mos1_T1_q=[-2.6859017682523882, -3.1425420089807976, -1.4457848495763397, -0.12098217319686988, 1.5591231516792479, -1.1179650176671911]
  global WP28_Mos1_T1_p=p[-.797474355081, -.433499999926, -.557075373677, .001359819885, -3.134982637669, -.011778030769]
  global WP28_Mos1_T1_q=[-2.5820856692233756, -3.149498109624623, -1.3870045692560584, -0.17380572227945468, 1.5587024486119303, -1.0142387662645218]
  global WP29_Mos1_T1_p=p[-.797492456394, -.530499999926, -.557045820837, .001318101491, -3.134975610626, -.011740131727]
  global WP29_Mos1_T1_q=[-2.4884120405871264, -3.162956038080441, -1.303240615969881, -0.24502012208909996, 1.5583785127547929, -0.9205816845508439]
  global WP30_Mos1_T1_p=p[-.517499999987, -.336499999991, -.557030058285, .001231290151, -3.134979369855, -.011758407393]
  global WP30_Mos1_T1_q=[-2.4575572915085644, -3.197660843308779, -1.882493548737708, 0.3686105560245027, 1.5601139590218063, -0.889078603208449]
  global WP31_Mos1_T1_p=p[-.517502976166, -.433499999926, -.557035222542, .001230636921, -3.134980586306, -.011748433550]
  global WP31_Mos1_T1_q=[-2.3276805517043337, -3.173415278609056, -1.8271387345445103, 0.28771963604773504, 1.5599652407630793, -0.7592858509756217]
  global WP32_Mos1_T1_p=p[-.517480949173, -.530499999926, -.557048298945, .001275948722, -3.135016509812, -.011783530471]
  global WP32_Mos1_T1_q=[-2.2224524802947947, -3.1511207047562273, -1.7493669028752254, 0.186576291832074, 1.559874434642144, -0.6541907179510416]
  global WP1_Mos1_T2_p=p[-.997999999689, .539016220973, -.392446493936, -3.134044553770, -.000802162574, .010540111149]
  global WP1_Mos1_T2_q=[-3.359404564391774, -3.042490735996984, -1.0527953393792764, -0.608435065567785, 1.561402029843705, 1.350721692910802]
  global WP2_Mos1_T2_p=p[-.998000000008, .442031451763, -.392394298559, -3.134033126020, -.000701372897, .010619585093]
  global WP2_Mos1_T2_q=[-3.267771807959933, -3.009495231907087, -1.1491152714815218, -0.5456321515909135, 1.560895057937787, 1.4424345387524724]
  global WP3_Mos1_T2_p=p[-.998000000000, .345034815000, -.392452392528, -3.134033581419, -.000520633556, .010337629383]
  global WP3_Mos1_T2_q=[-3.1724406920363823, -2.987946503565221, -1.2157226601719886, -0.5014184792475378, 1.560347370623711, 1.5378974682480917]
  global WP4_Mos1_T2_p=p[-.717999999690, .539017262991, -.392441236741, -3.134022090059, -.000628080714, .010487726859]
  global WP4_Mos1_T2_q=[-3.4355156803060267, -2.879849839776805, -1.6734325818067077, -0.15004424066949618, 1.5636190024998275, 1.2749422911988249]
  global WP5_Mos1_T2_p=p[-.714941794435, .442015470243, -.392452778378, -3.134075239889, -.000599492624, .010521606476]
  global WP5_Mos1_T2_q=[-3.3150319121226377, -2.8706641541376223, -1.7617752065865009, -0.07157272277964033, 1.5629360332111886, 1.395507536005914]
  global WP6_Mos1_T2_p=p[-.716036123132, .345011785381, -.392423502659, -3.133976777631, -.000614872850, .010553790430]
  global WP6_Mos1_T2_q=[-3.1841957342340184, -2.867712315068786, -1.8201182388288464, -0.017035645501089824, 1.5620313749708863, 1.5263830655533612]
  global WP7_Mos1_T2_p=p[-.539892765790, .447529829769, -.394334082832, -2.221673587755, 2.220359747494, .016075893585]
  global WP7_Mos1_T2_q=[-3.508436565143349, -2.8778408153141295, -1.6885341156561058, -0.1364212878921922, 1.5642828412814556, -3.51054729152684]
  global WP8_Mos1_T2_p=p[-.441999999822, .447516902268, -.394370526309, -2.221671983872, 2.220470984058, .015923084613]
  global WP8_Mos1_T2_q=[-3.5579894791114293, -2.8677793088683528, -1.83968666735883, 0.004824235428806365, 1.5652926959286058, -3.559925371716014]
  global WP9_Mos1_T2_p=p[-.993174238061, .247999177551, -.392406744722, -3.134045104847, -.000622748340, .010504693600]
  global WP9_Mos1_T2_q=[-3.0745771474123367, -2.971499798619117, -1.2687169756682115, -0.4655119085056878, 1.5598502373401748, 1.6357110373141075]
  global WP10_Mos1_T2_p=p[-.997999999632, .151019854922, -.392380256015, -3.134026135470, -.000653018074, .010483422378]
  global WP10_Mos1_T2_q=[-2.9770253479632367, -2.9706426724609765, -1.271099810289119, -0.46480640456241495, 1.5592731296496292, 1.7332483872142173]
  global WP11_Mos1_T2_p=p[-.997465570729, .054006583850, -.392352209754, -3.134040357902, -.000699596910, .010618336885]
  global WP11_Mos1_T2_q=[-2.8804451329614453, -2.9730005871641856, -1.2628031737759127, -0.4715059140483202, 1.5587650959230965, 1.829801338037113]
  global WP12_Mos1_T2_p=p[-.717999999658, .248015944423, -.392359082158, -3.134047049747, -.000633327238, .010620647253]
  global WP12_Mos1_T2_q=[-3.0482081331701587, -2.867156858459104, -1.8540466444803014, 0.015331771448991827, 1.5613083249405033, 1.662392941308017]
  global WP13_Mos1_T2_p=p[-.717938842046, .151002710304, -.392371757792, -3.134082862494, -.000694366291, .010543443133]
  global WP13_Mos1_T2_q=[-2.9112362409696, -2.867157355488098, -1.868297042714385, 0.028377508304319773, 1.5606452195075902, 1.7993444689458074]
  global WP14_Mos1_T2_p=p[-.718000000508, .054019247217, -.392375928997, -3.134083099030, -.000707344255, .010605999399]
  global WP14_Mos1_T2_q=[-2.7783575823675224, -2.866746439819643, -1.8590653208981394, 0.017560812616782384, 1.5600375699657878, 1.9322115136833973]
  global WP15_Mos1_T2_p=p[-.539999999727, .145502720074, -.394337539870, -2.221672944466, 2.220424624019, .016045244686]
  global WP15_Mos1_T2_q=[-3.0986310649563764, -2.86925118025588, -1.9081151893669563, 0.07197636287428266, 1.5617250799626807, -3.1005234100612205]
  global WP16_Mos1_T2_p=p[-.441999999763, .145510565920, -.394331010142, -2.221603678469, 2.220532858942, .016025984168]
  global WP16_Mos1_T2_q=[-3.0911280694437036, -2.8970598463942197, -2.064129697960582, 0.2557496031837781, 1.5621856361030424, -3.0927378991455923]
  global WP17_Mos1_T2_p=p[-.998000001553, -.043078773174, -.394375735881, .002005777421, -3.134683736801, -.011724575049]
  global WP17_Mos1_T2_q=[-3.0637251129672807, -2.9743975643768037, -1.258658182546366, -0.4725699546838884, 1.55979621877471, -1.495914914385704]
  global WP18_Mos1_T2_p=p[-.998000000941, -.139977273322, -.394447207121, .001818859707, -3.134760497001, -.011725527604]
  global WP18_Mos1_T2_q=[-2.9660233497063815, -2.9707068144223636, -1.2707573978879942, -0.46504603655828447, 1.5592618727286567, -1.3980862863903116]
  global WP19_Mos1_T2_p=p[-.998000006604, -.237011040712, -.394397701083, .001861192392, -3.134680859974, -.011767949565]
  global WP19_Mos1_T2_q=[-2.8698577188551835, -2.974315387167465, -1.258240991837118, -0.47472970526409064, 1.5587019013178685, -1.3019462070113228]
  global WP20_Mos1_T2_p=p[-.717617572395, -.043016871811, -.394330230086, .001902149342, -3.134629387176, -.011711792614]
  global WP20_Mos1_T2_q=[-3.0325625714388686, -2.8669796491649, -1.8572970132553976, 0.01844872137970724, 1.561263725052996, -1.4643607143490005]
  global WP21_Mos1_T2_p=p[-.718000005932, -.139987475107, -.394309700148, .001819148691, -3.134589051982, -.011678721065]
  global WP21_Mos1_T2_q=[-2.895962314260531, -2.866911342694423, -1.8681645356924284, 0.028122314744165877, 1.5605513086812481, -1.3276927282348705]
  global WP22_Mos1_T2_p=p[-.717999997821, -.236995125284, -.394313440010, .001822531137, -3.134509615755, -.011739244240]
  global WP22_Mos1_T2_q=[-2.7638084864017505, -2.866465935156254, -1.856411075130108, 0.014764792919493076, 1.5598717733809615, -1.1955470548030886]
  global WP23_Mos1_T2_p=p[-.540000001025, -.134477951721, -.394366218139, -2.221585327980, 2.220450671258, .015993774363]
  global WP23_Mos1_T2_q=[-2.6912908320714153, -2.8687468475135716, -1.9114976016330134, 0.07115085091663785, 1.5598015187987513, -2.693112334617004]
  global WP24_Mos1_T2_p=p[-.441999999497, -.134521631992, -.394334595861, -2.221683022150, 2.220490897867, .015974580155]
  global WP24_Mos1_T2_q=[-2.6170634210490644, -2.8970784738749997, -2.067786771690699, 0.2551254294864259, 1.5601389792576794, -2.618704935498167]
  global WP25_Mos1_T2_p=p[-.998000004873, -.331015955029, -.394372253957, .001781124345, -3.134648238273, -.011760817390]
  global WP25_Mos1_T2_q=[-2.7799231638351056, -2.98532128451383, -1.2221106113455331, -0.5006555783713607, 1.5582242498539396, -1.2119634286800078]
  global WP26_Mos1_T2_p=p[-.998000001755, -.430974952066, -.394415299260, .001816191599, -3.134692190068, -.011794210973]
  global WP26_Mos1_T2_q=[-2.689226173322936, -3.0063698567539587, -1.1563756248301083, -0.5462630505098671, 1.5577556193069564, -1.1212948600055546]
  global WP27_Mos1_T2_p=p[-.997999998008, -.527983626148, -.394343174025, .001804729555, -3.134626077203, -.011702787479]
  global WP27_Mos1_T2_q=[-2.607064401157514, -3.037854737930423, -1.0632092061177447, -0.6086689914949384, 1.557346745858276, -1.0391335276494154]
  global WP28_Mos1_T2_p=p[-.718000001665, -.334013716754, -.394333974689, .001773925742, -3.134599453894, -.011672540008]
  global WP28_Mos1_T2_q=[-2.640572526821882, -2.866460878634188, -1.8214009332896879, -0.02151227398524025, 1.5594492936483975, -1.0723047325025918]
  global WP29_Mos1_T2_p=p[-.718000005828, -.430991318158, -.394328971330, .001728773842, -3.134588437276, -.011690849752]
  global WP29_Mos1_T2_q=[-2.529094100852158, -2.8689753260925093, -1.7634918197626295, -0.07801856908542248, 1.5590374321103786, -0.9608382385011343]
  global WP30_Mos1_T2_p=p[-.718000004396, -.527967839075, -.394279637216, .001653916998, -3.134505619227, -.011677447350]
  global WP30_Mos1_T2_q=[-2.4305003370480556, -2.8768151140993576, -1.6828309596886122, -0.1517732011304469, 1.5586605363336015, -0.8622474437149226]
  global WP31_Mos1_T2_p=p[-.540000000724, -.436526285425, -.394330128273, -2.221736444272, 2.220519424622, .016011475106]
  global WP31_Mos1_T2_q=[-2.3528331827871636, -2.874893584844574, -1.6986873029412068, -0.1387678931789944, 1.5587673191579874, -2.3548523177454515]
  global WP32_Mos1_T2_p=p[-.440842117491, -.436537013456, -.394295632573, -2.221831087126, 2.220433070247, .016005961427]
  global WP32_Mos1_T2_q=[-2.254010519840117, -2.8654602752069898, -1.8520568374581892, 0.004169165599297507, 1.5593145831948327, -2.255982717183918]
  def Inicializacion():
    $ 32 "Inicializacion" "noBreak"
    $ 33 "Inicializacion"
    $ 34 "MoveJ"
    $ 35 "Arranque" "breakAfter"
    movej(pose_add(get_target_tcp_pose(), pose_sub(Arranque_to_p, Arranque_from_p)), a=1.3962634015954636, v=1.0471975511965976)
    $ 36 "Init Herramienta"
    $ 37 "StepCode = 1"
    StepCode = 1
    $ 38 "If ManoConCarton"
    if (ManoConCarton):
      $ 44 "ManoConCarton = False"
      ManoConCarton = False
      $ 45 "If NCapaAct[linea-1]≟1 and NMovAct[linea-1]≟1"
      if (NCapaAct[linea-1] == 1 and NMovAct[linea-1] == 1):
        $ 46 "CartonBase[linea-1] = True"
        CartonBase[linea-1] = True
      else:
        $ 47 "Else" "noBreak"
        $ 48 "NCapaAct[linea-1] = NCapaAct[linea-1] + 1"
        NCapaAct[linea-1] = NCapaAct[linea-1] + 1
        $ 49 "NMovAct[linea-1] = 1"
        NMovAct[linea-1] = 1
      end
      $ 50 "PonerCarton[linea-1] = False"
      PonerCarton[linea-1] = False
    end
    $ 51 "If ManoConProd"
    if (ManoConProd):
      $ 52 "ManoConProd = request_boolean_from_primary_client('¡Atención! Robot con producto. ¿Quieres continuar?')"
      ManoConProd = request_boolean_from_primary_client("¡Atención! Robot con producto. ¿Quieres continuar?")
    end
    $ 53 "If ManoConProd or ManoConCarton"
    if (ManoConProd or ManoConCarton):
      $ 54 "Per_LineaDeshab=True"
      Per_LineaDeshab=True
    else:
      $ 55 "Else" "noBreak"
      $ 56 "oEV1 =  False "
      oEV1 =   False
      $ 58 "Wait: 0.5"
      sleep(0.5)
      $ 59 "payload = PesoTool"
      payload = PesoTool
      $ 60 "set_payload(payload,cog_vacio)"
      set_payload(payload,cog_vacio)
    end
    $ 62 "Rutina Home"
    $ 63 "StepCode = 2"
    StepCode = 2
    $ 64 "actual = get_actual_tcp_pose()"
    actual = get_actual_tcp_pose()
    $ 65 "If actual[2] < 430/1000"
    if (actual[2] < 430/1000):
      $ 66 "actual[2] = 430/1000"
      actual[2] = 430/1000
      $ 67 "movel(actual,0.5,0.25,0,0)"
      movel(actual,0.5,0.25,0,0)
      $ 68 "actual = get_actual_tcp_pose()"
      actual = get_actual_tcp_pose()
    end
    $ 69 "If actual[1] > -400/1000"
    if (actual[1] > -400/1000):
      $ 70 "actual[1] = -400/1000"
      actual[1] = -400/1000
      $ 71 "movel(actual,0.5,0.25,0,0)"
      movel(actual,0.5,0.25,0,0)
    end
    $ 72 "movej(Home_q,0.5,0.25,0,0)"
    movej(Home_q,0.5,0.25,0,0)
    $ 76 "If ManoConProd ≟ False "
    if (ManoConProd  ==   False  ):
      $ 77 "Script: Calculos_previos.script"
      global PCogida = PuntosCogida[Programa-1]
      global OffsetZPreCogida = 50
      global PPreCogida = PCogida
      global zPCogida = (AltoTransporte - AltoBaseRobot)/1000 + Rec_AltoPrd[Programa-1]/1000 - 3/1000 - 13/1000
      global zPPreCogida = zPCogida + OffsetZPreCogida/1000
      PPreCogida[2] = zPPreCogida
      #PPreCogida[2] = zPPreCogida - pos_bajada[linea-1]/1000
      $ 78 "MoveJTrans(PPreCogida,Base_const,0.5,0.5,0,0)"
      MoveJTrans(PPreCogida,p[0.0,0.0,0.0,0.0,0.0,0.0],0.5,0.5,0,0)
    else:
      $ 79 "Else" "noBreak"
      $ 80 "Script: Calculos_previos.script"
      global PCogida = PuntosCogida[Programa-1]
      global OffsetZPreCogida = 50
      global PPreCogida = PCogida
      global zPCogida = (AltoTransporte - AltoBaseRobot)/1000 + Rec_AltoPrd[Programa-1]/1000 - 3/1000 - 13/1000
      global zPPreCogida = zPCogida + OffsetZPreCogida/1000
      PPreCogida[2] = zPPreCogida
      #PPreCogida[2] = zPPreCogida - pos_bajada[linea-1]/1000
      $ 81 "Script: Continuar.script"
      global PContinuar = Home_p

      local rpy = rotvec2rpy([PCogida[3],PCogida[4],PCogida[5]])
      rpy[0]=3.142
      rpy[1]=0
      local rotvec = rpy2rotvec(rpy)
      PContinuar[3] = rotvec[0]
      PContinuar[4] = rotvec[1]
      PContinuar[5] = rotvec[2]
      $ 82 "movej(PContinuar,0.5,0.25,0,0)"
      movej(PContinuar,0.5,0.25,0,0)
    end
    $ 83 "If NCapaAct[linea-1]>Rec_NCapasTot[Programa_1-1]"
    if (NCapaAct[linea-1]>Rec_NCapasTot[Programa_1-1]):
      $ 84 "StepCode = 3"
      StepCode = 3
      $ 85 "palet_completo(linea-1)"
      palet_completo(linea-1)
      $ 86 "popup('Check de seguridad. Número de capa mayor que el número de capas totales. Dando palet completo...',title='Aviso', warning = True, error = False, blocking = False)"
      popup("Check de seguridad. Número de capa mayor que el número de capas totales. Dando palet completo...",title="Aviso", warning = True, error = False, blocking = False)
    end
  end
  def Calculos():
    $ 87 "Calculos" "noBreak"
    $ 88 "Calculos"
    $ 89 "StepCode = 10"
    StepCode = 10
    $ 90 "If pos_bajada[linea_ant-1]<pos_bajada[linea-1] and linea_ant≠linea and ManoConProd≟ False "
    if (pos_bajada[linea_ant-1]<pos_bajada[linea-1]  and  linea_ant != linea  and  ManoConProd ==   False  ):
      $ 91 "pos_bajada[linea-1]=pos_bajada[linea_ant-1]"
      pos_bajada[linea-1]=pos_bajada[linea_ant-1]
    end
    $ 92 "Script: Calculos.script"
    ##########################COGIDA##########################

    #get_pos	#Selección del punto de cogida

    global PCogida = PuntosCogida[Programa_1-1]

    #get_xy

    global PPreCogida = PCogida
    global PPerchCogida = PCogida
    global PPostCogida = PCogida
    #PPaso2 es un punto de paso para que cuando se coja el producto se de la señal de ProdListo = False en cuanto sube la altura del producto
    global PPaso2 = PCogida

    #get_z #NO USAMOS BASE DE COGIDA

    #Offsets Z de cogida

    global OffsetZPreCogida = 50
    global OffsetZPerchCogida = 320
    global OffsetZPostCogida = 320

    if (Rec_AltoPrd[Programa_1-1] > OffsetZPostCogida):
    	OffsetZPerchCogida = Rec_AltoPrd[Programa_1-1] + 20
    	OffsetZPostCogida = Rec_AltoPrd[Programa_1-1] + 20
    end

    #Ajustes manuales es por la compresión de las ventosas
    global zPCogida = (AltoTransporte - AltoBaseRobot)/1000 + Rec_AltoPrd[Programa_1-1]/1000  - 3/1000 - 13/1000# los ultimos 11 son por la ventosa
    global zPPreCogida = zPCogida + OffsetZPreCogida/1000
    global zPPerchCogida = zPCogida + OffsetZPerchCogida/1000
    global zPPostCogida = zPPerchCogida



    ##########################DEJADA##########################

    #Selección del plano de dejada
    #Tenemos que modificar los planos de dejada para que funcionen independientemente y poder ajustar el mosaico al centro del palet independientemente de la linea que sea#RGR 30/11/22#
    global wObjDejada2 = pose_trans(wObjDejadaRef,p[0,0,0,0,0,0])
    global wObjDejada1 = pose_trans(wObjDejadaRef,p[0,-0.708 - AnchoPalet/1000,0,0,0,0])


    #global wObjDejada2 = wObjDejadaRef
    #global wObjDejada1 = pose_trans(wObjDejada2,p[0,-0.708 - AnchoPalet/1000,0,0,0,0])

    global wObjDejada = [wObjDejada1, wObjDejada2]
    global wObjDejadaAct = wObjDejada[linea-1]
    wObjDejadaAct[2] = -AltoBaseRobot/1000 + AltoPalet/1000


    #get_pos #Selección del punto de dejada

    if Rec_TipoCapa[NCapaAct[linea-1]-1] == 1:

       global PDejada = P_Tipo1[NMovAct[linea-1]-1]

    elif Rec_TipoCapa[NCapaAct[linea-1]-1] == 2:

       global PDejada = P_Tipo2[NMovAct[linea-1]-1]

    end

    #Anular rotaciones en X e Y
    local rpy = rotvec2rpy([PDejada[3],PDejada[4],PDejada[5]])
    rpy[0]=3.142
    rpy[1]=0
    local rotvec = rpy2rotvec(rpy)
    PDejada[3] = rotvec[0]
    PDejada[4] = rotvec[1]
    PDejada[5] = rotvec[2]


    global yPPerchDejada = yPPerchDejada_min
    if yPPerchDejada>0.3:
        yPPerchDejada = 0.3
    end
    if linea == 1:
        yPPerchDejada = yPPerchDejada_max
        if yPPerchDejada <0.5:
             yPPerchDejada = 0.5
        end
    end

    if xPPerchDejada>0.3:
        xPPerchDejada = 0.3
    end

    #get_xy
    global PPreDejada = PDejada
    global PPreDejada2 = PDejada
    global PPerchDejada = p[-200,0,0,PDejada[3],PDejada[4],PDejada[5]]
    global PPostDejada = PDejada
    #global PPreDejada1 = PDejada  ##CambioRubén##

    #get_aprox
    if linea == 2:
    		global aprox = 1
    elif linea == 1:
    		global aprox = 7
    end

    PPerchDejada[0] = xPPerchDejada - Offset/1000*cos(aprox*3.1415/4)
    PPerchDejada[1] = yPPerchDejada - Offset/1000*sin(aprox*3.1415/4)
    PPreDejada[0] = PPreDejada[0] - Offset/1000*cos(aprox*3.1415/4)
    PPreDejada[1] = PPreDejada[1] - Offset/1000*sin(aprox*3.1415/4)

    #get_z

    #Offsets Z de dejada
    global OffsetZPreDejada = 50
    global OffsetZPerchDejada = 90
    global OffsetZPostDejada = 50
    #global OffsetZPreDejada1 = zaprox[Programa_1] ##CambioRubén##

    global zPDejada = (NCapaAct[linea-1]*Rec_AltoPrd[Programa_1-1])/1000 + 10/1000 # los 10mm de margen de la ventosa
    global zPPreDejada = zPDejada + OffsetZPreDejada/1000
    global zPPerchDejada = zPDejada + OffsetZPerchDejada/1000
    global zPPostDejada = zPDejada + OffsetZPostDejada/1000
    #glogal zPPreDejada1 = zPDejada + OffsetZPreDejada1/1000 ##CambioRubén##

    #Equiparación de Perchs/Posts
    if zPPerchCogida < zPPerchDejada + wObjDejadaAct[2]:
                   zPPerchCogida = zPPerchDejada + wObjDejadaAct[2]
                   zPPostCogida = zPPerchCogida
    else:
                   zPPerchDejada = zPPerchCogida + norm(wObjDejadaAct[2])
    end

    #Actualizar z´s (incluyendo si está entrando en juego la columna)
    PDejada[2] = zPDejada - pos_bajada[linea-1]/1000
    PPreDejada[2] = zPPreDejada - pos_bajada[linea-1]/1000
    #PPreDejada1[2] = zPPreDejada1 - pos_bajada[linea-1]/1000 ##CambioRubén##
    PPreDejada2[2] = PPreDejada[2]
    PPerchDejada[2] = zPPerchDejada - pos_bajada[linea-1]/1000
    PPostDejada[2] = zPPostDejada - pos_bajada[linea-1]/1000

    PCogida[2] = zPCogida - pos_bajada[linea-1]/1000
    PPreCogida[2] = zPPreCogida - pos_bajada[linea-1]/1000
    PPaso2[2] = zPCogida + OffsetZPerchCogida/1000 - pos_bajada[linea-1]/1000
    PPostCogida[2] = zPPostCogida - pos_bajada[linea-1]/1000
    PPerchCogida[2] = PPostCogida[2]

    ##########################CARTÓN##########################
    #PPerchCogidaCarton es el punto bueno para liberar
    global PPerchCogidaCarton = PPerchCogidaCar_p
    global PCogidaCarton = PCogidaCarton_p

    PPerchCogidaCarton[2] = PPerchCogidaCarton[2] - pos_bajada[linea-1]/1000
    PCogidaCarton[2] = PCogidaCarton[2] - pos_bajada[linea-1]/1000

    pos_objetivo = PCogidaCarton


    global PDejadaCarton = pose_trans(Pbf, PDejadaCarton_p)
    global PPreDejadaCarton = PDejadaCarton
    global PPerchDejadaCarton = PDejadaCarton

    if Rec_Carton[0] and NCapaAct[linea-1] == 1 and NMovAct[linea-1] == 1 and not(CartonBase[linea-1]):

    	PonerCarton[linea-1] = True
    	PDejada[2] = 0
    end


    ##########################COLUMNA##########################

    #if ConfigRbt[1] == True   #Añadido RGR 24/11/2022#
    #
    #	#Obtengo coordenadas de los puntos mas críticos respecto de la base
    #	#Recordar que no tengo base de cogida
    #	#Actualizo pos_subida para subir a partir de pos_bajada
    #	pos_subida[linea-1] = pos_bajada[linea-1]
    #
    #
    #	#Me aseguro que de voy a llegar a los puntos críticos (PPostCogida y PPostDejada) (respecto a la base porque es el alcance real del robot).
    #	#Si no llego, voy subiendo columna (en un escalón de ajuste_col mm) y quitando esto a los puntos hasta que sea capaz de llegar
    #	local PPostDejada_base = pose_trans(wObjDejadaAct,PPostDejada)
    #	local PPostDejada_seguridad = PPostDejada_base
    #	PPostDejada_seguridad[2] = PPostDejada_base[2] + 0.13 #añado 15 cm de seguridad adicional (para que no jure bandera)
    #
    #	#PPostDejada_seguridad[2] = PPostDejada_base[2]
    #
    #	local PPostCogida_seguridad = PPostCogida
    #	PPostCogida_seguridad[2] = PPostCogida[2] + 0.13
    #
    #	#PPostCogida_seguridad[2] = PPostCogida[2]
    #
    #	if is_within_safety_limits(PPostDejada_seguridad) == False or is_within_safety_limits(PPostCogida_seguridad) == False:
    #    	local ajuste_col = 10
    #    	while is_within_safety_limits(PPostDejada_seguridad) == False or is_within_safety_limits(PPostCogida_seguridad) == False :
    #	         pos_subida[linea-1] = pos_subida[linea-1] + ajuste_col
    #	         PPostCogida_seguridad[2] = PPostCogida_seguridad[2] - ajuste_col/1000
    #	         PPostDejada_seguridad[2] = PPostDejada_seguridad[2] - ajuste_col/1000
    #	         sleep(0.01)
    #	    end
    #
    #		#Actualizo alturas
    #	    #para la Cogida no actualizar el plano nunca, porque afectaría al punto de cogida tb. Y sólo queremos cambiar Perch y Post!
    #		PPostCogida[2] = zPPostCogida - pos_subida[linea-1]/1000
    #		PPerchCogida[2] = PPostCogida[2]
    #
    #	              #PPerchCogidaCarton[2] = PPostCogida[2]
    #
    #
    #	    #para la dejada sí se podría actualizar el plano en lugar de todos los puntos
    #		PDejada[2] = zPDejada - pos_subida[linea-1]/1000
    #		PPreDejada[2] = zPPreDejada - pos_subida[linea-1]/1000
    #	               PPreDejada2[2] = PPreDejada[2]
    #		PPerchDejada[2] = zPPerchDejada - pos_subida[linea-1]/1000
    #		PPostDejada[2] = zPPostDejada - pos_subida[linea-1]/1000
    #	end
    #
    #
    #	PDejadaCarton[2] = PDejada[2]
    #
    #	PPerchDejadaCarton[0] = PDejadaCarton[0] - 1015/1000
    #	PPerchDejadaCarton[2] = PPerchDejada[2]
    #
    #	PPreDejadaCarton[2] = PDejadaCarton[2] + 50/1000
    #
    #	if linea == 1:
    #		local rpy = rotvec2rpy([PPerchDejadaCarton[3],PPerchDejadaCarton[4],PPerchDejadaCarton[5]])
    #		rpy[2]=rpy[2] - d2r(15)#15
    #		local rotvec = rpy2rotvec(rpy)
    #		PPerchDejadaCarton[3] = rotvec[0]
    #		PPerchDejadaCarton[4] = rotvec[1]
    #		PPerchDejadaCarton[5] = rotvec[2]
    #	end
    #
    #
    #
    #	#CHECK DE SEGURIDAD
    #	if pos_subida[linea-1] > 900:
    #		StepCode = 99
    #		pop_up("Altura columna inalcanzable para este movimiento. Contacta al servicio técnico",3 ,True)
    #	end
    #end 		#Añadido RGR 24/11/2022#


    ##########################EVITAR SEVILLANAS##########################

    #ESTANDARIZAR PUNTO COGIDA

    #Obtengo el valor de la rotación del punto de cogida respecto del plano de dejada para evaluar hacia dónde tengo que girar y evitar sevillanas
    global PCogida_plano = pose_trans(Pbf,PCogida)
    rpy = rotvec2rpy([PCogida_plano[3],PCogida_plano[4],PCogida_plano[5]])
    global RZ_PCogida = r2d(rpy[2])

    global RZ_PCogida_bis = 180

    if RZ_PCogida >= -45 and RZ_PCogida <= 45:
    	RZ_PCogida_bis = 0
    end

    if RZ_PCogida > -135 and RZ_PCogida < -45:
    	RZ_PCogida_bis = -90
    end

    if RZ_PCogida > 45 and RZ_PCogida < 135:
    	RZ_PCogida_bis = 90
    end


    #ESTANDARIZAR PUNTO DEJADA
    rpy = rotvec2rpy([PDejada[3],PDejada[4],PDejada[5]])
    global RZ_PDejada = r2d(rpy[2])

    global RZ_PDejada_bis = 180

    if RZ_PDejada >= -45 and RZ_PDejada <= 45:
    	RZ_PDejada_bis = 0
    end

    if RZ_PDejada > -135 and RZ_PDejada < -45:
    	RZ_PDejada_bis = -90
    end

    if RZ_PDejada > 45 and RZ_PDejada < 135:
    	RZ_PDejada_bis = 90
    end

    #sumo una constante para que sean todos positivos y sacar la diferencia

    global diferencia = (RZ_PDejada_bis + 90) - (RZ_PCogida_bis + 90)


    global RZ_PPaso3 = 90 + RZ_PCogida
    #-

    if diferencia >= -45 and diferencia <= 45:
    	RZ_PPaso3 = 0 + RZ_PCogida
    end

    if diferencia > -135 and diferencia < -45:
    	RZ_PPaso3 = -90 + RZ_PCogida
    end

    if diferencia > 45 and diferencia < 135:
    	RZ_PPaso3 = 90 + RZ_PCogida
    end


    rpy[2] = d2r(RZ_PPaso3)
    local rotvec = rpy2rotvec(rpy)


    if linea == 1:
    	global PPaso3 = p[0,(800 + 150)/1000,PPerchDejada[2], rotvec[0], rotvec[1], rotvec[2]]
                  #if NCapaAct[linea-1] < 4:
                           #  PDejada[2] = PDejada[2] -10/1000
                  #else:
                           #  PDejada[2] = PDejada[2] - 10/1000
                  #end
    else:
    	global PPaso3 = p[0,(0 + 150)/1000,PPerchDejada[2], rotvec[0], rotvec[1], rotvec[2]]
    end
  end
  def Movimientos():
    $ 93 "Movimientos" "noBreak"
    $ 94 "Movimientos"
    $ 95 "If LineaHabilitada[linea-1] or Per_LineaDeshab"
    if (LineaHabilitada[linea-1]  or  Per_LineaDeshab):
      $ 96 "Per_LineaDeshab= False "
      Per_LineaDeshab=  False
      $ 97 "If ManoConProd≟ False and not(PonerCarton[linea-1])"
      if (ManoConProd ==   False  and not(PonerCarton[linea-1])):
        $ 98 "Cogida"
        $ 99 "StepCode = 11"
        StepCode = 11
        $ 100 "MoveJTrans(PPreCogida,Base_const,2,2,0,0)"
        MoveJTrans(PPreCogida,p[0.0,0.0,0.0,0.0,0.0,0.0],2,2,0,0)
        $ 105 "MoveLTrans(PCogida,Base_const,0.5,0.25,0,0)"
        MoveLTrans(PCogida,p[0.0,0.0,0.0,0.0,0.0,0.0],0.5,0.25,0,0)
        $ 106 "If Rec_Cogida2en2[Programa_1-1]"
        if (Rec_Cogida2en2[Programa_1-1]):
          $ 107 "If Movs2en2[NMovAct[linea-1]-1]"
          if (Movs2en2[NMovAct[linea-1]-1]):
            $ 110 "ContPrd = 0"
            ContPrd = 0
            $ 111 "payload = PesoTool + 2*Rec_PesoPrd[Programa_1-1]"
            payload = PesoTool + 2*Rec_PesoPrd[Programa_1-1]
            $ 112 "cog = [0/1000,0/1000,(Rec_AltoPrd[Programa_1-1]/2)/1000]"
            cog = [0/1000,0/1000,(Rec_AltoPrd[Programa_1-1]/2)/1000]
            $ 113 "set_payload(payload, cog)"
            set_payload(payload, cog)
            $ 114 "Wait: 0.5"
            sleep(0.5)
          else:
            $ 116 "Else" "noBreak"
            $ 119 "ContPrd = 1"
            ContPrd = 1
            $ 120 "payload = PesoTool + Rec_PesoPrd[Programa_1-1]"
            payload = PesoTool + Rec_PesoPrd[Programa_1-1]
            $ 121 "cog = [0/1000,0/1000,(Rec_AltoPrd[Programa_1-1]/2)/1000]"
            cog = [0/1000,0/1000,(Rec_AltoPrd[Programa_1-1]/2)/1000]
            $ 122 "set_payload(payload, cog)"
            set_payload(payload, cog)
            $ 124 "Wait: 0.5"
            sleep(0.5)
          end
        else:
          $ 125 "Else" "noBreak"
          $ 126 "If Rec_2Vacios[Programa_1-1]"
          if (Rec_2Vacios[Programa_1-1]):
            $ 129 "payload = PesoTool + Rec_PesoPrd[Programa_1-1]"
            payload = PesoTool + Rec_PesoPrd[Programa_1-1]
            $ 130 "cog = [0/1000,0/1000,70/1000 + (Rec_AltoPrd[Programa_1-1]/2)/1000]"
            cog = [0/1000,0/1000,70/1000 + (Rec_AltoPrd[Programa_1-1]/2)/1000]
            $ 131 "set_payload(payload, cog)"
            set_payload(payload, cog)
            $ 133 "Wait: 0.5"
            sleep(0.5)
          else:
            $ 134 "Else" "noBreak"
            $ 135 "oEV1 =  True "
            oEV1 =   True
            $ 137 "payload = PesoTool + Rec_PesoPrd[Programa_1-1]"
            payload = PesoTool + Rec_PesoPrd[Programa_1-1]
            $ 138 "cog = [0/1000,0/1000,0/1000 + (Rec_AltoPrd[Programa_1-1]/2)/1000]"
            cog = [0/1000,0/1000,0/1000 + (Rec_AltoPrd[Programa_1-1]/2)/1000]
            $ 139 "set_payload(payload, cog)"
            set_payload(payload, cog)
            $ 141 "Wait: 0.5"
            sleep(0.5)
          end
          $ 142 "ContPrd = 0"
          ContPrd = 0
        end
        $ 143 "ManoConProd = True"
        ManoConProd = True
        $ 144 "Set Permiso_off=Apagar"
        set_configurable_digital_out(5, False)
      end
      $ 153 "If ManoConProd and not(PonerCarton[linea-1])"
      if (ManoConProd and not(PonerCarton[linea-1])):
        $ 154 "Dejada"
        $ 155 "StepCode = 12"
        StepCode = 12
        $ 156 "Actualización bajada columna"
        $ 157 "If NMovAct[linea-1] ≟ Rec_NMovsCapa[Programa_1-1] and Rec_Carton[NCapaAct[linea-1]]"
        if (NMovAct[linea-1]  ==  Rec_NMovsCapa[Programa_1-1] and Rec_Carton[NCapaAct[linea-1]]):
          $ 158 "If pos_subida[linea-1]>425"
          if (pos_subida[linea-1]>425):
            $ 159 "pos_bajada[linea-1]=425"
            pos_bajada[linea-1]=425
          else:
            $ 160 "Else" "noBreak"
            $ 161 "pos_bajada[linea-1]=pos_subida[linea-1]"
            pos_bajada[linea-1]=pos_subida[linea-1]
          end
        else:
          $ 162 "Else" "noBreak"
          $ 163 "If pos_subida[linea-1]>umbral_bajada"
          if (pos_subida[linea-1]>umbral_bajada):
            $ 164 "pos_bajada[linea-1]=umbral_bajada"
            pos_bajada[linea-1]=umbral_bajada
          else:
            $ 165 "Else" "noBreak"
            $ 166 "pos_bajada[linea-1]=pos_subida[linea-1]"
            pos_bajada[linea-1]=pos_subida[linea-1]
          end
        end
        $ 167 "PPreCogida[2] = zPCogida + OffsetZPreCogida/1000 - pos_bajada[linea-1]/1000"
        PPreCogida[2] = zPCogida + OffsetZPreCogida/1000 - pos_bajada[linea-1]/1000
        $ 168 "Wait PalletOk[linea-1]"
        while (not(PalletOk[linea-1])):
          sync()
        end
        $ 171 "'##Probar el script de MoveL o el movimiento convencionar al punto de dejada Segura y ver si funciona correctamente'"
        # '##Probar el script de MoveL o el movimiento convencionar al punto de dejada Segura y ver si funciona correctamente'
        $ 173 "MoveJ"
        $ 174 "PDejadaSegura" "breakAfter"
        movej(get_inverse_kin(PDejadaSegura_p, qnear=PDejadaSegura_q), a=1.3962634015954636, v=1.0471975511965976)
        $ 175 "MoveL"
        $ 176 "If linea≟2"
        if (linea == 2):
          $ 177 "Punto_de_paso_1" "breakAfter"
          movel(Punto_de_paso_1_p, a=1.2, v=0.9)
        else:
          $ 178 "ElseIf linea≟1"
          if (linea == 1):
            $ 179 "Punto_de_paso_2" "breakAfter"
            movel(Punto_de_paso_2_p, a=1.2, v=0.9)
          end
        end
        $ 181 "MoveLTrans(PPreDejada,wObjDejadaAct,1,1,0,0.01)"
        MoveLTrans(PPreDejada,wObjDejadaAct,1,1,0,0.01)
        $ 183 "'MovL preDejada1 añadido por Rubén (movimieno de dejada en z final von altura modificable en variable zaprox[])'"
        # 'MovL preDejada1 añadido por Rubén (movimieno de dejada en z final von altura modificable en variable zaprox[])'
        $ 185 "MoveLTrans(PDejada,wObjDejadaAct,0.5,0.5,0,0)"
        MoveLTrans(PDejada,wObjDejadaAct,0.5,0.5,0,0)
        $ 186 "oEV1=  False "
        oEV1=   False
        $ 188 "payload = PesoTool"
        payload = PesoTool
        $ 189 "set_payload(payload,cog_vacio)"
        set_payload(payload,cog_vacio)
        $ 191 "Wait: 0.75"
        sleep(0.75)
        $ 192 "ManoConProd = False"
        ManoConProd = False
        $ 193 "If NMovAct[linea-1]≟Rec_NMovsCapa[Programa_1-1] and Rec_Carton[NCapaAct[linea-1]]"
        if (NMovAct[linea-1] == Rec_NMovsCapa[Programa_1-1] and Rec_Carton[NCapaAct[linea-1]]):
          $ 194 "PonerCarton[linea-1] = True"
          PonerCarton[linea-1] = True
        else:
          $ 197 "ElseIf NMovAct[linea-1]≟Rec_NMovsCapa[Programa_1-1]"
          if (NMovAct[linea-1] == Rec_NMovsCapa[Programa_1-1]):
            $ 198 "NCapaAct[linea-1] = NCapaAct[linea-1] + 1"
            NCapaAct[linea-1] = NCapaAct[linea-1] + 1
            $ 199 "NMovAct[linea-1] = 1"
            NMovAct[linea-1] = 1
          else:
            $ 200 "Else" "noBreak"
            $ 201 "NMovAct[linea-1] =NMovAct[linea-1] + 1"
            NMovAct[linea-1] =NMovAct[linea-1] + 1
          end
        end
        $ 202 "If NCapaAct[linea-1]>Rec_NCapasTot[Programa_1-1]"
        if (NCapaAct[linea-1]>Rec_NCapasTot[Programa_1-1]):
          $ 203 "palet_completo(linea-1)"
          palet_completo(linea-1)
          $ 204 "CartonBase[linea-1] = False"
          CartonBase[linea-1] = False
          $ 205 "PPreCogida[2] = zPCogida + OffsetZPreCogida/1000 - pos_bajada[linea-1]/1000"
          PPreCogida[2] = zPCogida + OffsetZPreCogida/1000 - pos_bajada[linea-1]/1000
        end
        $ 206 "MoveLTrans(PPostDejada,wObjDejadaAct,1,1,0,0.025)"
        MoveLTrans(PPostDejada,wObjDejadaAct,1,1,0,0.025)
        $ 207 "MoveL"
        $ 208 "If linea≟2"
        if (linea == 2):
          $ 209 "Punto_de_paso_1" "breakAfter"
          movel(Punto_de_paso_1_p, a=1.2, v=0.9)
        else:
          $ 210 "Else" "noBreak"
          $ 211 "Punto_de_paso_2" "breakAfter"
          movel(Punto_de_paso_2_p, a=1.2, v=0.9)
        end
        $ 214 "MoveJTrans(PPreCogida,Base_const,2,2,0,0)"
        MoveJTrans(PPreCogida,p[0.0,0.0,0.0,0.0,0.0,0.0],2,2,0,0)
      end
    end
  end
  def CargarDatos():
    $ 485 "CargarDatos" "noBreak"
    $ 486 "StepCode = 9"
    StepCode = 9
    $ 487 "If  False "
    if (  False  ):
      $ 488 "MoveJ"
      $ 489 "Home" "breakAfter"
      movej(Home_q, a=1.3962634015954636, v=1.0471975511965976)
      $ 490 "PDejadaSegura" "breakAfter"
      movej(PDejadaSegura_q, a=1.3962634015954636, v=1.0471975511965976)
      $ 491 "PPerchCogidaCar" "breakAfter"
      movej(PPerchCogidaCar_q, a=1.3962634015954636, v=1.0471975511965976)
      $ 492 "PCogidaCarton" "breakAfter"
      movej(PCogidaCarton_q, a=1.3962634015954636, v=1.0471975511965976)
      $ 493 "PDejadaCarton" "breakAfter"
      movej(PDejadaCarton_q, a=1.3962634015954636, v=1.0471975511965976)
      $ 494 "Punto_de_paso_1" "breakAfter"
      movej(Punto_de_paso_1_q, a=1.3962634015954636, v=1.0471975511965976)
      $ 495 "Punto_de_paso_2" "breakAfter"
      movej(Punto_de_paso_2_q, a=1.3962634015954636, v=1.0471975511965976)
      $ 496 "PIntermedio" "breakAfter"
      movej(PIntermedio_q, a=1.3962634015954636, v=1.0471975511965976)
    end
    $ 497 "Puntos de cogida"
    $ 498 "If  False "
    if (  False  ):
      $ 499 "'Forma de definir poses moviendo el robot'"
      # 'Forma de definir poses moviendo el robot'
      $ 500 "MoveJ"
      $ 501 "PCogida_P1" "breakAfter"
      movej(get_inverse_kin(PCogida_P1_p, qnear=PCogida_P1_q), a=1.3962634015954636, v=1.0471975511965976)
    end
    $ 502 "Mosaicos"
    $ 503 "If Rec_Mosaico[Programa_1-1]≟1"
    if (Rec_Mosaico[Programa_1-1] == 1):
      $ 504 "Mosaico1"
      $ 505 "If  False "
      if (  False  ):
        $ 506 "'Forma de definir poses moviendo el robot'"
        # 'Forma de definir poses moviendo el robot'
        $ 507 "Puntos capa tipo 1"
        $ 508 "MoveJ"
        $ 509 "WP1_Mos1_T1" "breakAfter"
        movej(get_inverse_kin(WP1_Mos1_T1_p, qnear=WP1_Mos1_T1_q), a=1.3962634015954636, v=1.0471975511965976)
        $ 510 "WP2_Mos1_T1" "breakAfter"
        movej(get_inverse_kin(WP2_Mos1_T1_p, qnear=WP2_Mos1_T1_q), a=1.3962634015954636, v=1.0471975511965976)
        $ 511 "WP3_Mos1_T1" "breakAfter"
        movej(get_inverse_kin(WP3_Mos1_T1_p, qnear=WP3_Mos1_T1_q), a=1.3962634015954636, v=1.0471975511965976)
        $ 512 "WP4_Mos1_T1" "breakAfter"
        movej(get_inverse_kin(WP4_Mos1_T1_p, qnear=WP4_Mos1_T1_q), a=1.3962634015954636, v=1.0471975511965976)
        $ 513 "WP5_Mos1_T1" "breakAfter"
        movej(get_inverse_kin(WP5_Mos1_T1_p, qnear=WP5_Mos1_T1_q), a=1.3962634015954636, v=1.0471975511965976)
        $ 514 "WP6_Mos1_T1" "breakAfter"
        movej(get_inverse_kin(WP6_Mos1_T1_p, qnear=WP6_Mos1_T1_q), a=1.3962634015954636, v=1.0471975511965976)
        $ 515 "WP7_Mos1_T1" "breakAfter"
        movej(get_inverse_kin(WP7_Mos1_T1_p, qnear=WP7_Mos1_T1_q), a=1.3962634015954636, v=1.0471975511965976)
        $ 516 "WP8_Mos1_T1" "breakAfter"
        movej(get_inverse_kin(WP8_Mos1_T1_p, qnear=WP8_Mos1_T1_q), a=1.3962634015954636, v=1.0471975511965976)
        $ 517 "WP9_Mos1_T1" "breakAfter"
        movej(get_inverse_kin(WP9_Mos1_T1_p, qnear=WP9_Mos1_T1_q), a=1.3962634015954636, v=1.0471975511965976)
        $ 518 "WP10_Mos1_T1" "breakAfter"
        movej(get_inverse_kin(WP10_Mos1_T1_p, qnear=WP10_Mos1_T1_q), a=1.3962634015954636, v=1.0471975511965976)
        $ 519 "WP11_Mos1_T1" "breakAfter"
        movej(get_inverse_kin(WP11_Mos1_T1_p, qnear=WP11_Mos1_T1_q), a=1.3962634015954636, v=1.0471975511965976)
        $ 520 "WP12_Mos1_T1" "breakAfter"
        movej(get_inverse_kin(WP12_Mos1_T1_p, qnear=WP12_Mos1_T1_q), a=1.3962634015954636, v=1.0471975511965976)
        $ 521 "WP13_Mos1_T1" "breakAfter"
        movej(get_inverse_kin(WP13_Mos1_T1_p, qnear=WP13_Mos1_T1_q), a=1.3962634015954636, v=1.0471975511965976)
        $ 522 "WP14_Mos1_T1" "breakAfter"
        movej(get_inverse_kin(WP14_Mos1_T1_p, qnear=WP14_Mos1_T1_q), a=1.3962634015954636, v=1.0471975511965976)
        $ 523 "WP15_Mos1_T1" "breakAfter"
        movej(get_inverse_kin(WP15_Mos1_T1_p, qnear=WP15_Mos1_T1_q), a=1.3962634015954636, v=1.0471975511965976)
        $ 524 "WP16_Mos1_T1" "breakAfter"
        movej(get_inverse_kin(WP16_Mos1_T1_p, qnear=WP16_Mos1_T1_q), a=1.3962634015954636, v=1.0471975511965976)
        $ 525 "WP17_Mos1_T1" "breakAfter"
        movej(get_inverse_kin(WP17_Mos1_T1_p, qnear=WP17_Mos1_T1_q), a=1.3962634015954636, v=1.0471975511965976)
        $ 526 "WP18_Mos1_T1" "breakAfter"
        movej(get_inverse_kin(WP18_Mos1_T1_p, qnear=WP18_Mos1_T1_q), a=1.3962634015954636, v=1.0471975511965976)
        $ 527 "WP19_Mos1_T1" "breakAfter"
        movej(get_inverse_kin(WP19_Mos1_T1_p, qnear=WP19_Mos1_T1_q), a=1.3962634015954636, v=1.0471975511965976)
        $ 528 "WP20_Mos1_T1" "breakAfter"
        movej(get_inverse_kin(WP20_Mos1_T1_p, qnear=WP20_Mos1_T1_q), a=1.3962634015954636, v=1.0471975511965976)
        $ 529 "WP21_Mos1_T1" "breakAfter"
        movej(get_inverse_kin(WP21_Mos1_T1_p, qnear=WP21_Mos1_T1_q), a=1.3962634015954636, v=1.0471975511965976)
        $ 530 "WP22_Mos1_T1" "breakAfter"
        movej(get_inverse_kin(WP22_Mos1_T1_p, qnear=WP22_Mos1_T1_q), a=1.3962634015954636, v=1.0471975511965976)
        $ 531 "WP23_Mos1_T1" "breakAfter"
        movej(get_inverse_kin(WP23_Mos1_T1_p, qnear=WP23_Mos1_T1_q), a=1.3962634015954636, v=1.0471975511965976)
        $ 532 "WP24_Mos1_T1" "breakAfter"
        movej(get_inverse_kin(WP24_Mos1_T1_p, qnear=WP24_Mos1_T1_q), a=1.3962634015954636, v=1.0471975511965976)
        $ 533 "WP25_Mos1_T1" "breakAfter"
        movej(get_inverse_kin(WP25_Mos1_T1_p, qnear=WP25_Mos1_T1_q), a=1.3962634015954636, v=1.0471975511965976)
        $ 534 "WP26_Mos1_T1" "breakAfter"
        movej(get_inverse_kin(WP26_Mos1_T1_p, qnear=WP26_Mos1_T1_q), a=1.3962634015954636, v=1.0471975511965976)
        $ 535 "WP27_Mos1_T1" "breakAfter"
        movej(get_inverse_kin(WP27_Mos1_T1_p, qnear=WP27_Mos1_T1_q), a=1.3962634015954636, v=1.0471975511965976)
        $ 536 "WP28_Mos1_T1" "breakAfter"
        movej(get_inverse_kin(WP28_Mos1_T1_p, qnear=WP28_Mos1_T1_q), a=1.3962634015954636, v=1.0471975511965976)
        $ 537 "WP29_Mos1_T1" "breakAfter"
        movej(get_inverse_kin(WP29_Mos1_T1_p, qnear=WP29_Mos1_T1_q), a=1.3962634015954636, v=1.0471975511965976)
        $ 538 "WP30_Mos1_T1" "breakAfter"
        movej(get_inverse_kin(WP30_Mos1_T1_p, qnear=WP30_Mos1_T1_q), a=1.3962634015954636, v=1.0471975511965976)
        $ 539 "WP31_Mos1_T1" "breakAfter"
        movej(get_inverse_kin(WP31_Mos1_T1_p, qnear=WP31_Mos1_T1_q), a=1.3962634015954636, v=1.0471975511965976)
        $ 540 "WP32_Mos1_T1" "breakAfter"
        movej(get_inverse_kin(WP32_Mos1_T1_p, qnear=WP32_Mos1_T1_q), a=1.3962634015954636, v=1.0471975511965976)
        $ 541 "Puntos capa tipo 2"
        $ 542 "MoveJ"
        $ 543 "WP1_Mos1_T2" "breakAfter"
        movej(get_inverse_kin(WP1_Mos1_T2_p, qnear=WP1_Mos1_T2_q), a=1.3962634015954636, v=1.0471975511965976)
        $ 544 "WP2_Mos1_T2" "breakAfter"
        movej(get_inverse_kin(WP2_Mos1_T2_p, qnear=WP2_Mos1_T2_q), a=1.3962634015954636, v=1.0471975511965976)
        $ 545 "WP3_Mos1_T2" "breakAfter"
        movej(get_inverse_kin(WP3_Mos1_T2_p, qnear=WP3_Mos1_T2_q), a=1.3962634015954636, v=1.0471975511965976)
        $ 546 "WP4_Mos1_T2" "breakAfter"
        movej(get_inverse_kin(WP4_Mos1_T2_p, qnear=WP4_Mos1_T2_q), a=1.3962634015954636, v=1.0471975511965976)
        $ 547 "WP5_Mos1_T2" "breakAfter"
        movej(get_inverse_kin(WP5_Mos1_T2_p, qnear=WP5_Mos1_T2_q), a=1.3962634015954636, v=1.0471975511965976)
        $ 548 "WP6_Mos1_T2" "breakAfter"
        movej(get_inverse_kin(WP6_Mos1_T2_p, qnear=WP6_Mos1_T2_q), a=1.3962634015954636, v=1.0471975511965976)
        $ 549 "WP7_Mos1_T2" "breakAfter"
        movej(get_inverse_kin(WP7_Mos1_T2_p, qnear=WP7_Mos1_T2_q), a=1.3962634015954636, v=1.0471975511965976)
        $ 550 "WP8_Mos1_T2" "breakAfter"
        movej(get_inverse_kin(WP8_Mos1_T2_p, qnear=WP8_Mos1_T2_q), a=1.3962634015954636, v=1.0471975511965976)
        $ 551 "WP9_Mos1_T2" "breakAfter"
        movej(get_inverse_kin(WP9_Mos1_T2_p, qnear=WP9_Mos1_T2_q), a=1.3962634015954636, v=1.0471975511965976)
        $ 552 "WP10_Mos1_T2" "breakAfter"
        movej(get_inverse_kin(WP10_Mos1_T2_p, qnear=WP10_Mos1_T2_q), a=1.3962634015954636, v=1.0471975511965976)
        $ 553 "WP11_Mos1_T2" "breakAfter"
        movej(get_inverse_kin(WP11_Mos1_T2_p, qnear=WP11_Mos1_T2_q), a=1.3962634015954636, v=1.0471975511965976)
        $ 554 "WP12_Mos1_T2" "breakAfter"
        movej(get_inverse_kin(WP12_Mos1_T2_p, qnear=WP12_Mos1_T2_q), a=1.3962634015954636, v=1.0471975511965976)
        $ 555 "WP13_Mos1_T2" "breakAfter"
        movej(get_inverse_kin(WP13_Mos1_T2_p, qnear=WP13_Mos1_T2_q), a=1.3962634015954636, v=1.0471975511965976)
        $ 556 "WP14_Mos1_T2" "breakAfter"
        movej(get_inverse_kin(WP14_Mos1_T2_p, qnear=WP14_Mos1_T2_q), a=1.3962634015954636, v=1.0471975511965976)
        $ 557 "WP15_Mos1_T2" "breakAfter"
        movej(get_inverse_kin(WP15_Mos1_T2_p, qnear=WP15_Mos1_T2_q), a=1.3962634015954636, v=1.0471975511965976)
        $ 558 "WP16_Mos1_T2" "breakAfter"
        movej(get_inverse_kin(WP16_Mos1_T2_p, qnear=WP16_Mos1_T2_q), a=1.3962634015954636, v=1.0471975511965976)
        $ 559 "WP17_Mos1_T2" "breakAfter"
        movej(get_inverse_kin(WP17_Mos1_T2_p, qnear=WP17_Mos1_T2_q), a=1.3962634015954636, v=1.0471975511965976)
        $ 560 "WP18_Mos1_T2" "breakAfter"
        movej(get_inverse_kin(WP18_Mos1_T2_p, qnear=WP18_Mos1_T2_q), a=1.3962634015954636, v=1.0471975511965976)
        $ 561 "WP19_Mos1_T2" "breakAfter"
        movej(get_inverse_kin(WP19_Mos1_T2_p, qnear=WP19_Mos1_T2_q), a=1.3962634015954636, v=1.0471975511965976)
        $ 562 "WP20_Mos1_T2" "breakAfter"
        movej(get_inverse_kin(WP20_Mos1_T2_p, qnear=WP20_Mos1_T2_q), a=1.3962634015954636, v=1.0471975511965976)
        $ 563 "WP21_Mos1_T2" "breakAfter"
        movej(get_inverse_kin(WP21_Mos1_T2_p, qnear=WP21_Mos1_T2_q), a=1.3962634015954636, v=1.0471975511965976)
        $ 564 "WP22_Mos1_T2" "breakAfter"
        movej(get_inverse_kin(WP22_Mos1_T2_p, qnear=WP22_Mos1_T2_q), a=1.3962634015954636, v=1.0471975511965976)
        $ 565 "WP23_Mos1_T2" "breakAfter"
        movej(get_inverse_kin(WP23_Mos1_T2_p, qnear=WP23_Mos1_T2_q), a=1.3962634015954636, v=1.0471975511965976)
        $ 566 "WP24_Mos1_T2" "breakAfter"
        movej(get_inverse_kin(WP24_Mos1_T2_p, qnear=WP24_Mos1_T2_q), a=1.3962634015954636, v=1.0471975511965976)
        $ 567 "WP25_Mos1_T2" "breakAfter"
        movej(get_inverse_kin(WP25_Mos1_T2_p, qnear=WP25_Mos1_T2_q), a=1.3962634015954636, v=1.0471975511965976)
        $ 568 "WP26_Mos1_T2" "breakAfter"
        movej(get_inverse_kin(WP26_Mos1_T2_p, qnear=WP26_Mos1_T2_q), a=1.3962634015954636, v=1.0471975511965976)
        $ 569 "WP27_Mos1_T2" "breakAfter"
        movej(get_inverse_kin(WP27_Mos1_T2_p, qnear=WP27_Mos1_T2_q), a=1.3962634015954636, v=1.0471975511965976)
        $ 570 "WP28_Mos1_T2" "breakAfter"
        movej(get_inverse_kin(WP28_Mos1_T2_p, qnear=WP28_Mos1_T2_q), a=1.3962634015954636, v=1.0471975511965976)
        $ 571 "WP29_Mos1_T2" "breakAfter"
        movej(get_inverse_kin(WP29_Mos1_T2_p, qnear=WP29_Mos1_T2_q), a=1.3962634015954636, v=1.0471975511965976)
        $ 572 "WP30_Mos1_T2" "breakAfter"
        movej(get_inverse_kin(WP30_Mos1_T2_p, qnear=WP30_Mos1_T2_q), a=1.3962634015954636, v=1.0471975511965976)
        $ 573 "WP31_Mos1_T2" "breakAfter"
        movej(get_inverse_kin(WP31_Mos1_T2_p, qnear=WP31_Mos1_T2_q), a=1.3962634015954636, v=1.0471975511965976)
        $ 574 "WP32_Mos1_T2" "breakAfter"
        movej(get_inverse_kin(WP32_Mos1_T2_p, qnear=WP32_Mos1_T2_q), a=1.3962634015954636, v=1.0471975511965976)
      end
      $ 575 "Script: mosaico1.script_bak_bak"
      #MOSAICO 1
      #P_Tipo1 y P_Tipo2 tienen que venir ya relativizados del asistente!

      if ModificarMos == True:

      	P_Tipo1_Mos1 = P_Tipo1
      	P_Tipo2_Mos1 = P_Tipo2
      	ordenM1_T1 = orden_T1
      	ordenM1_T2 = orden_T2

      end

      ModificarMos = False

      P_Tipo1 = P_Tipo1_Mos1
      P_Tipo2 = P_Tipo2_Mos1


      #En caso de que actualice movimientos de 2 en 2 (modificación de mosaico o crear nuevo)
      if Cogida2en2 == True:

      	Movs2en2_M1_T1 = Movs2en2_Tipo1
      	Movs2en2_M1_T2 = Movs2en2_Tipo2

      end

      Cogida2en2 = False

      #Siempre, si hay algún movimiento doble, actualizo si el movimiento actual lo es o no
      if Rec_Cogida2en2[Programa_1-1] == True:
      	if Rec_TipoCapa[NCapaAct[linea-1]-1] == 1:
      		Movs2en2 = Movs2en2_M1_T1
      		if linea == 1:
      			Movs2en2[NMovAct[linea-1]-1] = Movs2en2[ordenM1_T1[NMovAct[linea-1]-1]-1]
      		end
      	else:
      		Movs2en2 = Movs2en2_M1_T2
      		if linea == 1:
      			Movs2en2[NMovAct[linea-1]-1] = Movs2en2[ordenM1_T2[NMovAct[linea-1]-1]-1]
      		end
      	end
      else:
      	Movs2en2[NMovAct[linea-1]-1] = False
      end

      if linea == 1:
          P_Tipo1[NMovAct[linea-1]-1] = P_Tipo1[ordenM1_T1[NMovAct[linea-1]-1]-1]
          P_Tipo2[NMovAct[linea-1]-1] = P_Tipo2[ordenM1_T2[NMovAct[linea-1]-1]-1]
      end
    else:
      $ 576 "ElseIf Rec_Mosaico[Programa_1-1]≟2"
      if (Rec_Mosaico[Programa_1-1] == 2):
        $ 577 "Mosaico2"
        $ 612 "Script: mosaico2.script_bak"
        #MOSAICO 2
        #P_Tipo1 y P_Tipo2 tienen que venir ya relativizados del asistente!

        if ModificarMos == True:

        	P_Tipo1_Mos2 = P_Tipo1
        	P_Tipo2_Mos2 = P_Tipo2
        	ordenM2_T1 = orden_T1
        	ordenM2_T2 = orden_T2

        end

        ModificarMos = False

        P_Tipo1 = P_Tipo1_Mos2
        P_Tipo2 = P_Tipo2_Mos2


        #En caso de que actualice movimientos de 2 en 2 (modificación de mosaico o crear nuevo)
        if Cogida2en2 == True:

        	Movs2en2_M2_T1 = Movs2en2_Tipo1
        	Movs2en2_M2_T2 = Movs2en2_Tipo2

        end

        Cogida2en2 = False

        #Siempre, si hay algún movimiento doble, actualizo si el movimiento actual lo es o no
        if Rec_Cogida2en2[Programa_1-1] == True:
        	if Rec_TipoCapa[NCapaAct[linea-1]-1] == 1:
        		Movs2en2 = Movs2en2_M2_T1
        		if linea == 1:
        			Movs2en2[NMovAct[linea-1]-1] = Movs2en2[ordenM2_T1[NMovAct[linea-1]-1]-1]
        		end
        	else:
        		Movs2en2 = Movs2en2_M2_T2
        		if linea == 1:
        			Movs2en2[NMovAct[linea-1]-1] = Movs2en2[ordenM2_T2[NMovAct[linea-1]-1]-1]
        		end
        	end
        else:
        	Movs2en2[NMovAct[linea-1]-1] = False
        end

        if linea == 1:
            P_Tipo1[NMovAct[linea-1]-1] = P_Tipo1[ordenM2_T1[NMovAct[linea-1]-1]-1]
            P_Tipo2[NMovAct[linea-1]-1] = P_Tipo2[ordenM2_T2[NMovAct[linea-1]-1]-1]
        end
      else:
        $ 613 "ElseIf Rec_Mosaico[Programa_1-1]≟3"
        if (Rec_Mosaico[Programa_1-1] == 3):
          $ 614 "Mosaico3"
          $ 660 "Script: mosaico3.script"
          #MOSAICO 3
          #P_Tipo1 y P_Tipo2 tienen que venir ya relativizados del asistente!

          if ModificarMos == True:

          	P_Tipo1_Mos3 = P_Tipo1
          	P_Tipo2_Mos3 = P_Tipo2
          	ordenM3_T1 = orden_T1
          	ordenM3_T2 = orden_T2

          end

          ModificarMos = False

          P_Tipo1 = P_Tipo1_Mos3
          P_Tipo2 = P_Tipo2_Mos3


          #En caso de que actualice movimientos de 2 en 2 (modificación de mosaico o crear nuevo)
          if Cogida2en2 == True:

          	Movs2en2_M3_T1 = Movs2en2_Tipo1
          	Movs2en2_M3_T2 = Movs2en2_Tipo2

          end

          Cogida2en2 = False

          #Siempre, si hay algún movimiento doble, actualizo si el movimiento actual lo es o no
          if Rec_Cogida2en2[Programa-1] == True:
          	if Rec_TipoCapa[NCapaAct[linea-1]-1] == 1:
          		Movs2en2 = Movs2en2_M3_T1
          		if linea == 1:
          			Movs2en2[NMovAct[linea-1]-1] = Movs2en2[ordenM3_T1[NMovAct[linea-1]-1]-1]
          		end
          	else:
          		Movs2en2 = Movs2en2_M3_T2
          		if linea == 1:
          			Movs2en2[NMovAct[linea-1]-1] = Movs2en2[ordenM3_T2[NMovAct[linea-1]-1]-1]
          		end
          	end
          else:
          	Movs2en2[NMovAct[linea-1]-1] = False
          end

          if linea == 1:
              P_Tipo1[NMovAct[linea-1]-1] = P_Tipo1[ordenM3_T1[NMovAct[linea-1]-1]-1]
              P_Tipo2[NMovAct[linea-1]-1] = P_Tipo2[ordenM3_T2[NMovAct[linea-1]-1]-1]
          end
        else:
          $ 661 "ElseIf Rec_Mosaico[Programa_1-1]≟4"
          if (Rec_Mosaico[Programa_1-1] == 4):
            $ 662 "Mosaico4"
            $ 668 "Script: mosaico4.script"
            #MOSAICO 4
            #P_Tipo1 y P_Tipo2 tienen que venir ya relativizados del asistente!

            if ModificarMos == True:

            	P_Tipo1_Mos4 = P_Tipo1
            	P_Tipo2_Mos4 = P_Tipo2
            	ordenM4_T1 = orden_T1
            	ordenM4_T2 = orden_T2

            end

            ModificarMos = False

            P_Tipo1 = P_Tipo1_Mos4
            P_Tipo2 = P_Tipo2_Mos4


            #En caso de que actualice movimientos de 2 en 2 (modificación de mosaico o crear nuevo)
            if Cogida2en2 == True:

            	Movs2en2_M4_T1 = Movs2en2_Tipo1
            	Movs2en2_M4_T2 = Movs2en2_Tipo2

            end

            Cogida2en2 = False

            #Siempre, si hay algún movimiento doble, actualizo si el movimiento actual lo es o no
            if Rec_Cogida2en2[Programa-1] == True:
            	if Rec_TipoCapa[NCapaAct[linea-1]-1] == 1:
            		Movs2en2 = Movs2en2_M4_T1
            		if linea == 1:
            			Movs2en2[NMovAct[linea-1]-1] = Movs2en2[ordenM4_T1[NMovAct[linea-1]-1]-1]
            		end
            	else:
            		Movs2en2 = Movs2en2_M4_T2
            		if linea == 1:
            			Movs2en2[NMovAct[linea-1]-1] = Movs2en2[ordenM4_T2[NMovAct[linea-1]-1]-1]
            		end
            	end
            else:
            	Movs2en2[NMovAct[linea-1]-1] = False
            end

            if linea == 1:
                P_Tipo1[NMovAct[linea-1]-1] = P_Tipo1[ordenM4_T1[NMovAct[linea-1]-1]-1]
                P_Tipo2[NMovAct[linea-1]-1] = P_Tipo2[ordenM4_T2[NMovAct[linea-1]-1]-1]
            end
          else:
            $ 669 "ElseIf Rec_Mosaico[Programa_1-1]≟5"
            if (Rec_Mosaico[Programa_1-1] == 5):
              $ 670 "Mosaico 5"
              $ 676 "Script: mosaico5.script"
              #MOSAICO 5
              #P_Tipo1 y P_Tipo2 tienen que venir ya relativizados del asistente!

              if ModificarMos == True:

              	P_Tipo1_Mos5 = P_Tipo1
              	P_Tipo2_Mos5 = P_Tipo2
              	ordenM5_T1 = orden_T1
              	ordenM5_T2 = orden_T2

              end

              ModificarMos = False

              P_Tipo1 = P_Tipo1_Mos5
              P_Tipo2 = P_Tipo2_Mos5


              #En caso de que actualice movimientos de 2 en 2 (modificación de mosaico o crear nuevo)
              if Cogida2en2 == True:

              	Movs2en2_M5_T1 = Movs2en2_Tipo1
              	Movs2en2_M5_T2 = Movs2en2_Tipo2

              end

              Cogida2en2 = False

              #Siempre, si hay algún movimiento doble, actualizo si el movimiento actual lo es o no
              if Rec_Cogida2en2[Programa-1] == True:
              	if Rec_TipoCapa[NCapaAct[linea-1]-1] == 1:
              		Movs2en2 = Movs2en2_M5_T1
              		if linea == 1:
              			Movs2en2[NMovAct[linea-1]-1] = Movs2en2[ordenM5_T1[NMovAct[linea-1]-1]-1]
              		end
              	else:
              		Movs2en2 = Movs2en2_M5_T2
              		if linea == 1:
              			Movs2en2[NMovAct[linea-1]-1] = Movs2en2[ordenM5_T2[NMovAct[linea-1]-1]-1]
              		end
              	end
              else:
              	Movs2en2[NMovAct[linea-1]-1] = False
              end

              if linea == 1:
                  P_Tipo1[NMovAct[linea-1]-1] = P_Tipo1[ordenM5_T1[NMovAct[linea-1]-1]-1]
                  P_Tipo2[NMovAct[linea-1]-1] = P_Tipo2[ordenM5_T2[NMovAct[linea-1]-1]-1]
              end
            else:
              $ 677 "ElseIf Rec_Mosaico[Programa_1-1]≟6"
              if (Rec_Mosaico[Programa_1-1] == 6):
                $ 678 "Mosaico 6"
                $ 684 "Script: mosaico6.script"
                #MOSAICO 6
                #P_Tipo1 y P_Tipo2 tienen que venir ya relativizados del asistente!

                if ModificarMos == True:

                	P_Tipo1_Mos6 = P_Tipo1
                	P_Tipo2_Mos6 = P_Tipo2
                	ordenM6_T1 = orden_T1
                	ordenM6_T2 = orden_T2

                end

                ModificarMos = False

                P_Tipo1 = P_Tipo1_Mos6
                P_Tipo2 = P_Tipo2_Mos6


                #En caso de que actualice movimientos de 2 en 2 (modificación de mosaico o crear nuevo)
                if Cogida2en2 == True:

                	Movs2en2_M6_T1 = Movs2en2_Tipo1
                	Movs2en2_M6_T2 = Movs2en2_Tipo2

                end

                Cogida2en2 = False

                #Siempre, si hay algún movimiento doble, actualizo si el movimiento actual lo es o no
                if Rec_Cogida2en2[Programa-1] == True:
                	if Rec_TipoCapa[NCapaAct[linea-1]-1] == 1:
                		Movs2en2 = Movs2en2_M6_T1
                		if linea == 1:
                			Movs2en2[NMovAct[linea-1]-1] = Movs2en2[ordenM6_T1[NMovAct[linea-1]-1]-1]
                		end
                	else:
                		Movs2en2 = Movs2en2_M6_T2
                		if linea == 1:
                			Movs2en2[NMovAct[linea-1]-1] = Movs2en2[ordenM6_T2[NMovAct[linea-1]-1]-1]
                		end
                	end
                else:
                	Movs2en2[NMovAct[linea-1]-1] = False
                end

                if linea == 1:
                    P_Tipo1[NMovAct[linea-1]-1] = P_Tipo1[ordenM6_T1[NMovAct[linea-1]-1]-1]
                    P_Tipo2[NMovAct[linea-1]-1] = P_Tipo2[ordenM6_T2[NMovAct[linea-1]-1]-1]
                end
              else:
                $ 685 "ElseIf Rec_Mosaico[Programa_1-1]≟7"
                if (Rec_Mosaico[Programa_1-1] == 7):
                  $ 686 "Mosaico 7"
                  $ 692 "Script: mosaico7.script"
                  #MOSAICO 7
                  #P_Tipo1 y P_Tipo2 tienen que venir ya relativizados del asistente!

                  if ModificarMos == True:

                  	P_Tipo1_Mos7 = P_Tipo1
                  	P_Tipo2_Mos7 = P_Tipo2
                  	ordenM7_T1 = orden_T1
                  	ordenM7_T2 = orden_T2

                  end

                  ModificarMos = False

                  P_Tipo1 = P_Tipo1_Mos7
                  P_Tipo2 = P_Tipo2_Mos7


                  #En caso de que actualice movimientos de 2 en 2 (modificación de mosaico o crear nuevo)
                  if Cogida2en2 == True:

                  	Movs2en2_M7_T1 = Movs2en2_Tipo1
                  	Movs2en2_M7_T2 = Movs2en2_Tipo2

                  end

                  Cogida2en2 = False

                  #Siempre, si hay algún movimiento doble, actualizo si el movimiento actual lo es o no
                  if Rec_Cogida2en2[Programa-1] == True:
                  	if Rec_TipoCapa[NCapaAct[linea-1]-1] == 1:
                  		Movs2en2 = Movs2en2_M7_T1
                  		if linea == 1:
                  			Movs2en2[NMovAct[linea-1]-1] = Movs2en2[ordenM7_T1[NMovAct[linea-1]-1]-1]
                  		end
                  	else:
                  		Movs2en2 = Movs2en2_M7_T2
                  		if linea == 1:
                  			Movs2en2[NMovAct[linea-1]-1] = Movs2en2[ordenM7_T2[NMovAct[linea-1]-1]-1]
                  		end
                  	end
                  else:
                  	Movs2en2[NMovAct[linea-1]-1] = False
                  end

                  if linea == 1:
                      P_Tipo1[NMovAct[linea-1]-1] = P_Tipo1[ordenM7_T1[NMovAct[linea-1]-1]-1]
                      P_Tipo2[NMovAct[linea-1]-1] = P_Tipo2[ordenM7_T2[NMovAct[linea-1]-1]-1]
                  end
                else:
                  $ 693 "ElseIf Rec_Mosaico[Programa_1-1]≟8"
                  if (Rec_Mosaico[Programa_1-1] == 8):
                    $ 694 "Mosaico 8"
                    $ 700 "Script: mosaico8.script"
                    #MOSAICO 8
                    #P_Tipo1 y P_Tipo2 tienen que venir ya relativizados del asistente!

                    if ModificarMos == True:

                    	P_Tipo1_Mos8 = P_Tipo1
                    	P_Tipo2_Mos8 = P_Tipo2
                    	ordenM8_T1 = orden_T1
                    	ordenM8_T2 = orden_T2

                    end

                    ModificarMos = False

                    P_Tipo1 = P_Tipo1_Mos8
                    P_Tipo2 = P_Tipo2_Mos8


                    #En caso de que actualice movimientos de 2 en 2 (modificación de mosaico o crear nuevo)
                    if Cogida2en2 == True:

                    	Movs2en2_M8_T1 = Movs2en2_Tipo1
                    	Movs2en2_M8_T2 = Movs2en2_Tipo2

                    end

                    Cogida2en2 = False

                    #Siempre, si hay algún movimiento doble, actualizo si el movimiento actual lo es o no
                    if Rec_Cogida2en2[Programa-1] == True:
                    	if Rec_TipoCapa[NCapaAct[linea-1]-1] == 1:
                    		Movs2en2 = Movs2en2_M8_T1
                    		if linea == 1:
                    			Movs2en2[NMovAct[linea-1]-1] = Movs2en2[ordenM8_T1[NMovAct[linea-1]-1]-1]
                    		end
                    	else:
                    		Movs2en2 = Movs2en2_M8_T2
                    		if linea == 1:
                    			Movs2en2[NMovAct[linea-1]-1] = Movs2en2[ordenM8_T2[NMovAct[linea-1]-1]-1]
                    		end
                    	end
                    else:
                    	Movs2en2[NMovAct[linea-1]-1] = False
                    end

                    if linea == 1:
                        P_Tipo1[NMovAct[linea-1]-1] = P_Tipo1[ordenM8_T1[NMovAct[linea-1]-1]-1]
                        P_Tipo2[NMovAct[linea-1]-1] = P_Tipo2[ordenM8_T2[NMovAct[linea-1]-1]-1]
                    end
                  else:
                    $ 701 "ElseIf Rec_Mosaico[Programa_1-1]≟9"
                    if (Rec_Mosaico[Programa_1-1] == 9):
                      $ 702 "Mosaico 9"
                      $ 708 "Script: mosaico9.script"
                      #MOSAICO 9
                      #P_Tipo1 y P_Tipo2 tienen que venir ya relativizados del asistente!

                      if ModificarMos == True:

                      	P_Tipo1_Mos9 = P_Tipo1
                      	P_Tipo2_Mos9 = P_Tipo2
                      	ordenM9_T1 = orden_T1
                      	ordenM9_T2 = orden_T2

                      end

                      ModificarMos = False

                      P_Tipo1 = P_Tipo1_Mos9
                      P_Tipo2 = P_Tipo2_Mos9


                      #En caso de que actualice movimientos de 2 en 2 (modificación de mosaico o crear nuevo)
                      if Cogida2en2 == True:

                      	Movs2en2_M9_T1 = Movs2en2_Tipo1
                      	Movs2en2_M9_T2 = Movs2en2_Tipo2

                      end

                      Cogida2en2 = False

                      #Siempre, si hay algún movimiento doble, actualizo si el movimiento actual lo es o no
                      if Rec_Cogida2en2[Programa-1] == True:
                      	if Rec_TipoCapa[NCapaAct[linea-1]-1] == 1:
                      		Movs2en2 = Movs2en2_M9_T1
                      		if linea == 1:
                      			Movs2en2[NMovAct[linea-1]-1] = Movs2en2[ordenM9_T1[NMovAct[linea-1]-1]-1]
                      		end
                      	else:
                      		Movs2en2 = Movs2en2_M9_T2
                      		if linea == 1:
                      			Movs2en2[NMovAct[linea-1]-1] = Movs2en2[ordenM9_T2[NMovAct[linea-1]-1]-1]
                      		end
                      	end
                      else:
                      	Movs2en2[NMovAct[linea-1]-1] = False
                      end

